// ---- FBs/Other Big Consumer/KNX/Linear/FB_OBC_Linear_KNX.TcPOU
FUNCTION_BLOCK FB_OBC_Linear_KNX
VAR_INPUT PERSISTENT
	bEnable									: BOOL;												//{#lynus.ag#()} //Enable the Fuctionblock and his logic
	bPowerDataInvers						: BOOL;												//With True its possible to invert all received power data from the electric meter
	bNoLinear								: BOOL;												//Output Power from the device is not linear. Use the Values from the Table Of Interpolation Points.
	diNrOfKNXMasterLine_IN					: DINT;												//Number of the KNX Master Function on what this function can receive or write data
	diNrOfEMS_IN							: DINT;												//Number of EMS what control this Device.
	diNrOfEM_IN_OBC							: DINT;												//Number of the electric meter for incoming power data. (Power Data for this Device)
	stSetupOBC								: ST_Setup_OBC;										//{#lynus.ag#()} //Setup other big consumer
	strGroupAddr							: EIB_GROUP_ADDR;									//KNX group address which should be controlled with this function
	arrTableOfInterpolationPoints			: ARRAY[1..10] OF REAL;								//Table Of Interpolation Points. Corresponds to the different power values in the non-linear curve of the device. The last value must correspond to the maximum power.
END_VAR
VAR_INPUT
END_VAR
VAR_OUTPUT
	stDataOBC								: ST_OBC_Output;									//{#lynus.ag#()} //Output Data other big consumer
	diNrOfOBC_OUT							: DINT;												//Active Number from the other big consumer for using on other functions
END_VAR
VAR
	{attribute 'hide'}
	fbOBC									: FB_BigConsumer;									//Function for other big consumer
	{attribute 'hide'}
	fbNumberDevice							: FB_NumberOfDevice;								//Function block to calcualte the number of the Device
	{attribute 'hide'}
	fbInterpolation							: FB_Lin_Interpolation;								//Function for interpolation
	fbDIExternalLock						: FB_XL1XXX_DI;										//Digital Input from external loock signal
	{attribute 'hide'}
	fbKNXSend								: EIB_2OCTET_FLOAT_SEND_EX;							//Function to send a Float value to the KNX Bus
	{attribute 'hide'}
	timDissableFunctions					: TON;												//Timer to dissable the Function after Lynus_Standards.Constants_General.tTimeDissableLynusFunctions Days without connection to the Lynus Cloud
	{attribute 'hide'}
	timResetConnectionOnGVL					: TON;												//Timer to try reset the connection Flag on the GVL. (When somebody delete the Connection Function and make only a onlinechange)
	{attribute 'hide'}
	arrPD									: ARRAY[1..27] OF FB_PersistentData_Number;			//Function to save persistent data 
	{attribute 'hide'}
	byWaitInStep							: BYTE;												//Wait in Step before start to clean data on PLC
	{attribute 'hide'}
	iStateGVLData							: INT;												//State machine to handle the data on the GVL
	{attribute 'hide'}
	diNumberOfActiveBatterys				: DINT;												//Number of active batterys
	{attribute 'hide'}
	diNumberOfBatteryInverterInEPO			: DINT;												//Number of battery inverters that work in Emergency Power operation 
	{attribute 'hide'}
	diCounterForGVL							: DINT;												//Counter to clean old data on GVL
	{attribute 'hide'}
	diLPForGVL								: DINT;												//Loop to clean old data on GVL
	{attribute 'hide'}
	dwSumSOC								: DWORD;											//Sum of the SOC from all batterys
	{attribute 'hide'}
	liLPBatteryData							: LINT;												//Loop to check some data from batterys
	{attribute 'hide'}
	liLPInEPO								: LINT;												//Loop to check if 1 or more battery inverters build a island grid	
END_VAR
VAR PERSISTENT
	{attribute 'conditionalshow'}
	diNrOfEMS_IN_CP							: DINT;												//Number of EMS what control this Device to compare with the original
END_VAR

//Creator : Kai Ebensperger
//Company : Lynus AG
//Date : 24.08.2021
//Version : 1.0.0.0

//With this function block its possible to control a other big consumer with the plc
//The output signal to control the big consumer is sending to the KNX Group Adress from the Inputs
//The value what is sending to the KNX Bus is between 0 and 100 to control the device.
//Also the Power Data can by displayed with this functionblock

//NOTE for diNr.....Designation => 
//_IN = Here Data come in from other Functions or go out to other functions about the GVL
//_OUT = Here Data go out to other functions about the GVL

(*------------------------------------------------------------Limits----------------------------------------------------------------------------------*)

diNrOfEMS_IN := LIMIT(0,diNrOfEMS_IN,Constants_Energy.diMaxNumberOfEMS);
	diNrOfEM_IN_OBC := LIMIT(0,diNrOfEM_IN_OBC,Constants_Energy.diMaxNumberOfElectricMeters);
		diNrOfKNXMasterLine_IN := LIMIT(0,diNrOfKNXMasterLine_IN,Constants_Bussystems.diMaxNumberOfKNXMasterKL6301);	

strGroupAddr.MAIN := LIMIT(0,strGroupAddr.MAIN,31);
	strGroupAddr.SUB_MAIN := LIMIT(0,strGroupAddr.SUB_MAIN,7);
			
(*------------------------------------------------------------------Power Data----------------------------------------------------------------------------*)

IF NOT bPowerDataInvers THEN
	fbOBC.lrCounterEnergyT1_Consumption := Lynus_Standards.GVL_Energy.stDataElectricMeters[diNrOfEM_IN_OBC].lrCounterEnergyT1_Production * 1000;
	fbOBC.lrCounterEnergyT2_Consumption := Lynus_Standards.GVL_Energy.stDataElectricMeters[diNrOfEM_IN_OBC].lrCounterEnergyT2_Production * 1000;
	fbOBC.lrCounterEnergyT1_Production := Lynus_Standards.GVL_Energy.stDataElectricMeters[diNrOfEM_IN_OBC].lrCounterEnergyT1_Consumption * 1000;
	fbOBC.lrCounterEnergyT2_Production := Lynus_Standards.GVL_Energy.stDataElectricMeters[diNrOfEM_IN_OBC].lrCounterEnergyT1_Consumption * 1000;
	fbOBC.lrTotalCounterEnergy_Consumption := Lynus_Standards.GVL_Energy.stDataElectricMeters[diNrOfEM_IN_OBC].lrTotalCounterEnergy_Production * 1000;
	fbOBC.lrTotalCounterEnergy_Production := Lynus_Standards.GVL_Energy.stDataElectricMeters[diNrOfEM_IN_OBC].lrTotalCounterEnergy_Consumption * 1000;
		fbOBC.lrPowerOBC := (Lynus_Standards.GVL_Energy.stDataElectricMeters[diNrOfEM_IN_OBC].lrPower * 1000) * - 1;
ELSE
	fbOBC.lrCounterEnergyT1_Consumption := Lynus_Standards.GVL_Energy.stDataElectricMeters[diNrOfEM_IN_OBC].lrCounterEnergyT1_Consumption * 1000;
	fbOBC.lrCounterEnergyT2_Consumption := Lynus_Standards.GVL_Energy.stDataElectricMeters[diNrOfEM_IN_OBC].lrCounterEnergyT2_Consumption * 1000;
	fbOBC.lrCounterEnergyT1_Production := Lynus_Standards.GVL_Energy.stDataElectricMeters[diNrOfEM_IN_OBC].lrCounterEnergyT1_Production * 1000;
	fbOBC.lrCounterEnergyT2_Production := Lynus_Standards.GVL_Energy.stDataElectricMeters[diNrOfEM_IN_OBC].lrCounterEnergyT2_Production * 1000;
	fbOBC.lrTotalCounterEnergy_Consumption := Lynus_Standards.GVL_Energy.stDataElectricMeters[diNrOfEM_IN_OBC].lrTotalCounterEnergy_Consumption * 1000;
	fbOBC.lrTotalCounterEnergy_Production := Lynus_Standards.GVL_Energy.stDataElectricMeters[diNrOfEM_IN_OBC].lrTotalCounterEnergy_Production * 1000;
		fbOBC.lrPowerOBC := Lynus_Standards.GVL_Energy.stDataElectricMeters[diNrOfEM_IN_OBC].lrPower * 1000;
END_IF

(*-------------------------------------------------------------Calcualte the number of OBC---------------------------------------------------------------*)

fbNumberDevice(
	diActualNumberOfDevices:= Lynus_Standards.GVL_Energy.stNumberOfDevices.diNumberOfOBC, 
	diMaxNumberOfDevices:= Constants_Energy.diMaxNumberOfOtherBigConsumers, 
	udiCounterOnlineChange:= TwinCAT_SystemInfoVarList._AppInfo.OnlineChangeCnt, 
	bNumberIsCalculatet=> , 
	bFPNumberIsCalculatet=> , 
	bOnlineChange=> , 
	diNumberForThisDevice=> diNrOfOBC_OUT, 
	diNumberOfTotalDevices=> );

//Write new Numer on GVL
IF fbNumberDevice.bFPNumberIsCalculatet THEN
	Lynus_Standards.GVL_Energy.stNumberOfDevices.diNumberOfOBC := fbNumberDevice.diNumberOfTotalDevices;	
END_IF 

//Delete old Number on GVL
IF fbNumberDevice.bOnlineChange THEN 
	Lynus_Standards.GVL_Energy.stNumberOfDevices.diNumberOfOBC := diNrOfOBC_OUT;	
		iStateGVLData := 1; 
END_IF

(*-------------------------------------------------------------Service from Backend is ready and check the connection to backen for dissabel/enable Function---------------------------------------------------------------*)

//Try to reset the variable for connection on the GVL. When all is normal then the Lynus Mqtt connection function set this variable to true in the next cycle
//When we have no connection to the backend then after Lynus_Standards.Constants_General.tTimeDissableLynusFunctions days the Function is dissabled with all of his functionalities
timResetConnectionOnGVL(IN:= NOT timResetConnectionOnGVL.Q, PT:= T#1H, Q=> , ET=> );
	IF timResetConnectionOnGVL.Q THEN Lynus_Standards.GVL_Communicator.bStateConnectionToEnableFunctions := FALSE; END_IF
		IF NOT Lynus_Standards.GVL_Communicator.bStateConnectionToEnableFunctions THEN timDissableFunctions.IN := TRUE; ELSE timDissableFunctions.IN := FALSE; END_IF  
			timDissableFunctions(IN:= , PT:= Lynus_Standards.Constants_General.tTimeDissableLynusFunctions, Q=> , ET=> );

(*------------------------------------------------------------------Error----------------------------------------------------------------------------*)

IF timDissableFunctions.Q THEN fbOBC.bWarning := TRUE; fbOBC.iWarningCode := 0; ELSE fbOBC.bWarning := FALSE; END_IF 
	IF Lynus_Standards.GVL_Energy.stNumberOfDevices.diNumberOfOBC > Constants_Energy.diMaxNumberOfOtherBigConsumers OR fbKNXSend.bError THEN 
		fbOBC.bError := TRUE;
	ELSE 
		fbOBC.bError := FALSE;
	END_IF 	
	
IF Lynus_Standards.GVL_Energy.stNumberOfDevices.diNumberOfOBC > Constants_Energy.diMaxNumberOfOtherBigConsumers THEN fbOBC.iErrorCode := 1;
ELSIF fbKNXSend.bError THEN fbOBC.iErrorCode := 0;
END_IF   	
	
(*------------------------------------------------------------------Logic----------------------------------------------------------------------------*)
	
//Calcualte the total SOC if we have more then 1 battery in our system
diNumberOfActiveBatterys := 0;
	dwSumSOC := 0;
		FOR liLPBatteryData := 1 TO Constants_Energy.diMaxNumberOfBatterys BY 1 DO
			IF Lynus_Standards.GVL_Energy.stDataOfBatterys[diNrOfEMS_IN,liLPBatteryData].bEnabled THEN diNumberOfActiveBatterys := diNumberOfActiveBatterys + 1; END_IF
				dwSumSOC := dwSumSOC + Lynus_Standards.GVL_Energy.stDataOfBatterys[diNrOfEMS_IN,liLPBatteryData].dwSOC;
		END_FOR
	
IF diNumberOfActiveBatterys > 0 THEN
	fbOBC.dwBatterySOC := DINT_TO_DWORD(DWORD_TO_DINT(dwSumSOC) / diNumberOfActiveBatterys);
ELSE
	fbOBC.dwBatterySOC := 100;	//When we have no battery in the ems system
END_IF

//Check if one or more Batterysystems or batteryinverter make island mode
diNumberOfBatteryInverterInEPO := 0;
	FOR liLPInEPO := 1 TO Constants_Energy.diMaxNumberOfBatteryInverters BY 1 DO
		IF Lynus_Standards.GVL_Energy.stDataOfBatteryInverters[diNrOfEMS_IN,liLPInEPO].bWorkOnIslandMode THEN fbOBC.bEPOIsActive := TRUE; diNumberOfBatteryInverterInEPO := diNumberOfBatteryInverterInEPO + 1; END_IF
	END_FOR 
		IF diNumberOfBatteryInverterInEPO <= 0 THEN fbOBC.bEPOIsActive := FALSE; END_IF

//Digital input for external lock signal
fbDIExternalLock(bInvers:= FALSE, bSignal=> );

fbOBC(
	bEnable:= bEnable AND NOT timDissableFunctions.Q,
	bError:= , 
	bEPOIsActive:= , 
	bExternalLock:= fbDIExternalLock.bSignal, 
	bWriteWithDelay:= TRUE, 
	iErrorCode:= , 
	iWarningCode:= , 
	dwBatterySOC:= , 
	lrTotalCounterEnergy_Consumption:= , 
	lrTotalCounterEnergy_Production:= , 
	lrCounterEnergyT1_Consumption:= , 
	lrCounterEnergyT2_Consumption:= , 
	lrCounterEnergyT1_Production:= , 
	lrCounterEnergyT2_Production:= , 
	lrPowerOBC:= , 
	rTargetPower:= Lynus_Standards.GVL_Energy.stDataOtherBigConsumers[diNrOfEMS_IN,diNrOfOBC_OUT].rTargetPowerEMS, 
	tTimDelayOutput:= T#5S, 
	stSetupOBC:= stSetupOBC, 
	stDataOBCOut=> , 
	stDataOBCOutDelay=> stDataOBC);											
	
(*-------------------------------------------------------------------------Output to KNX----------------------------------------------------------------------*)

IF bNoLinear THEN 
	fbInterpolation.rXInputValue := (stSetupOBC.rMaxPower * fbOBC.stDataOBCOut.rTargetPower) / 100; 
		fbInterpolation.arrYIntermediateValues[1] := 10;
			fbInterpolation.arrYIntermediateValues[2] := 20;
				fbInterpolation.arrYIntermediateValues[3] := 30;
					fbInterpolation.arrYIntermediateValues[4] := 40;
						fbInterpolation.arrYIntermediateValues[5] := 50;
	fbInterpolation.arrYIntermediateValues[6] := 60;
		fbInterpolation.arrYIntermediateValues[7] := 70;
			fbInterpolation.arrYIntermediateValues[8] := 80;
				fbInterpolation.arrYIntermediateValues[9] := 90;
					fbInterpolation.arrYIntermediateValues[10] := 100;
	fbInterpolation(rXInputValue:=, arrXIntermediateValues:= arrTableOfInterpolationPoints, arrYIntermediateValues:=, rYOutputValue=> );
END_IF

IF bNoLinear THEN 
	fbKNXSend.rData := fbInterpolation.rYOutputValue;
ELSE
	fbKNXSend.rData := fbOBC.stDataOBCOut.rTargetPower;
END_IF
	
fbKNXSend(
	bStart:= TRUE, 
	iMode:= 2, 
	CyclePolling:= T#200MS, 
	MinSendTime:= T#500MS, 
	Group_Address:= strGroupAddr, 
	rData:= , 
	str_Rec:= Lynus_Standards.GVL_Bussystems.stDataOfKNXMasterKL6301[diNrOfKNXMasterLine_IN], 
	bEnableReadReq:= FALSE, 
	bBusy=> , 
	bError=> , 
	iErrorID=> );

(*-----------------------------------------------------------Handle data to Global structure for the other big consumers-----------------------------------------------------------------*)

//Delte al old Data on GVL after a online change or change on the variable diNrOfEMS_IDOD
IF diNrOfEM_IN_OBC <> diNrOfEMS_IN_CP AND iStateGVLData = 0 THEN iStateGVLData := 10; END_IF 

CASE iStateGVLData OF
	
	0://Init Step
		byWaitInStep := 0;
			diCounterForGVL := 1;
	
	1://Wait for 4 Steps before clean al Data on GVL
		byWaitInStep := byWaitInStep + 1;
			IF byWaitInStep >= 4 AND fbNumberDevice.bNumberIsCalculatet THEN iStateGVLData := 2; END_IF
				//To much Devices, back to the Init step
				IF byWaitInStep >= 4 AND NOT fbNumberDevice.bNumberIsCalculatet THEN iStateGVLData := 0; END_IF	
			
	2://Clear all Data in GVL
		FOR diLPForGVL := 1 TO Constants_Energy.diMaxNumberOfEMS BY 1 DO 
			Lynus_Standards.GVL_Energy.stDataOtherBigConsumers[diLPForGVL,diCounterForGVL].bEnabled := FALSE;
				Lynus_Standards.GVL_Energy.stDataOtherBigConsumers[diLPForGVL,diCounterForGVL].bIsControllable := FALSE;
					Lynus_Standards.GVL_Energy.stDataOtherBigConsumers[diLPForGVL,diCounterForGVL].byPriority := 0;
						Lynus_Standards.GVL_Energy.stDataOtherBigConsumers[diLPForGVL,diCounterForGVL].byErrorWarning := 0;
							Lynus_Standards.GVL_Energy.stDataOtherBigConsumers[diLPForGVL,diCounterForGVL].lrPower := 0;
								Lynus_Standards.GVL_Energy.stDataOtherBigConsumers[diLPForGVL,diCounterForGVL].lrPowerConsumption := 0;
									Lynus_Standards.GVL_Energy.stDataOtherBigConsumers[diLPForGVL,diCounterForGVL].lrPowerProduction := 0;
										Lynus_Standards.GVL_Energy.stDataOtherBigConsumers[diLPForGVL,diCounterForGVL].rMaxPower := 0;
											//Set also the target value from ems back here to 0 and not in EMS function because EMS is in Standy when we have a online change (Problem when we delete a ems function and make a online change)
											Lynus_Standards.GVL_Energy.stDataOtherBigConsumers[diLPForGVL,diCounterForGVL].rTargetPowerEMS := 0;
		END_FOR
			diCounterForGVL := diCounterForGVL + 1;
				diCounterForGVL := LIMIT(0,diCounterForGVL,Constants_Energy.diMaxNumberOfOtherBigConsumers);
					//Back to the init step
					IF diCounterForGVL >= Constants_Energy.diMaxNumberOfOtherBigConsumers THEN iStateGVLData := 0; END_IF

	10://Clear old Data on GVL 	
		Lynus_Standards.GVL_Energy.stDataOtherBigConsumers[diNrOfEMS_IN_CP,diNrOfOBC_OUT].bEnabled := FALSE;
			Lynus_Standards.GVL_Energy.stDataOtherBigConsumers[diNrOfEMS_IN_CP,diNrOfOBC_OUT].bIsControllable := FALSE;
				Lynus_Standards.GVL_Energy.stDataOtherBigConsumers[diNrOfEMS_IN_CP,diNrOfOBC_OUT].byPriority := 0;
					Lynus_Standards.GVL_Energy.stDataOtherBigConsumers[diNrOfEMS_IN_CP,diNrOfOBC_OUT].byErrorWarning := 0;
						Lynus_Standards.GVL_Energy.stDataOtherBigConsumers[diNrOfEMS_IN_CP,diNrOfOBC_OUT].lrPower := 0;
							Lynus_Standards.GVL_Energy.stDataOtherBigConsumers[diNrOfEMS_IN_CP,diNrOfOBC_OUT].lrPowerConsumption := 0;
								Lynus_Standards.GVL_Energy.stDataOtherBigConsumers[diNrOfEMS_IN_CP,diNrOfOBC_OUT].lrPowerProduction := 0;
									Lynus_Standards.GVL_Energy.stDataOtherBigConsumers[diNrOfEMS_IN_CP,diNrOfOBC_OUT].rMaxPower := 0;
	
		diNrOfEMS_IN_CP := diNrOfEMS_IN;
			//Back to the init step
			iStateGVLData := 0;

END_CASE 	 

IF diNrOfOBC_OUT > 0 AND fbNumberDevice.bNumberIsCalculatet AND diNrOfEMS_IN > 0 THEN
	Lynus_Standards.GVL_Energy.stDataOtherBigConsumers[diNrOfEMS_IN,diNrOfOBC_OUT].bEnabled := fbOBC.stDataOBCOut.bEnabled;
		Lynus_Standards.GVL_Energy.stDataOtherBigConsumers[diNrOfEMS_IN,diNrOfOBC_OUT].bIsControllable := TRUE;
			Lynus_Standards.GVL_Energy.stDataOtherBigConsumers[diNrOfEMS_IN,diNrOfOBC_OUT].byPriority := fbOBC.stDataOBCOut.byPriority;
				Lynus_Standards.GVL_Energy.stDataOtherBigConsumers[diNrOfEMS_IN,diNrOfOBC_OUT].byErrorWarning := fbOBC.stDataOBCOut.byErrorWarning;
					Lynus_Standards.GVL_Energy.stDataOtherBigConsumers[diNrOfEMS_IN,diNrOfOBC_OUT].lrPower := fbOBC.stDataOBCOut.lrPower;
						Lynus_Standards.GVL_Energy.stDataOtherBigConsumers[diNrOfEMS_IN,diNrOfOBC_OUT].lrPowerConsumption := fbOBC.stDataOBCOut.lrPowerConsumption;
							Lynus_Standards.GVL_Energy.stDataOtherBigConsumers[diNrOfEMS_IN,diNrOfOBC_OUT].lrPowerProduction := fbOBC.stDataOBCOut.lrPowerProduction;
								Lynus_Standards.GVL_Energy.stDataOtherBigConsumers[diNrOfEMS_IN,diNrOfOBC_OUT].rMaxPower := fbOBC.stDataOBCOut.rMaxPower;
END_IF

(*----------------------------------------------------------Save persistent data----------------------------------------------------------------*)

arrPD[1](lrValue:= BOOL_TO_LREAL(bEnable), bEventBasedActive=> );
arrPD[2](lrValue:= BOOL_TO_LREAL(bPowerDataInvers), bEventBasedActive=> );
arrPD[3](lrValue:= DINT_TO_LREAL(diNrOfEMS_IN), bEventBasedActive=> );
arrPD[4](lrValue:= DINT_TO_LREAL(diNrOfEM_IN_OBC), bEventBasedActive=> );
arrPD[5](lrValue:= DINT_TO_LREAL(diNrOfEMS_IN_CP), bEventBasedActive=> );
arrPD[6](lrValue:= BOOL_TO_LREAL(stSetupOBC.bManualyOn), bEventBasedActive=> );
arrPD[7](lrValue:= BOOL_TO_LREAL(stSetupOBC.bOnEmergPowerOff), bEventBasedActive=> );
arrPD[8](lrValue:= BYTE_TO_LREAL(stSetupOBC.byDisableSOC), bEventBasedActive=> );
arrPD[9](lrValue:= BYTE_TO_LREAL(stSetupOBC.byEnableSOC), bEventBasedActive=> );
arrPD[10](lrValue:= BYTE_TO_LREAL(stSetupOBC.byManualyTargetPower), bEventBasedActive=> );
arrPD[11](lrValue:= BYTE_TO_LREAL(stSetupOBC.byPriority), bEventBasedActive=> );
arrPD[12](lrValue:= REAL_TO_LREAL(stSetupOBC.rMaxPower), bEventBasedActive=> );
arrPD[13](lrValue:= DINT_TO_LREAL(diNrOfKNXMasterLine_IN), bEventBasedActive=> );
arrPD[14](lrValue:= BYTE_TO_LREAL(strGroupAddr.MAIN), bEventBasedActive=> );
arrPD[15](lrValue:= BYTE_TO_LREAL(strGroupAddr.NUMBER), bEventBasedActive=> );
arrPD[16](lrValue:= BYTE_TO_LREAL(strGroupAddr.SUB_MAIN), bEventBasedActive=> );
arrPD[17](lrValue:= BOOL_TO_LREAL(bNoLinear), bEventBasedActive=> );
arrPD[18](lrValue:= REAL_TO_LREAL(arrTableOfInterpolationPoints[1]), bEventBasedActive=> );
arrPD[19](lrValue:= REAL_TO_LREAL(arrTableOfInterpolationPoints[2]), bEventBasedActive=> );
arrPD[20](lrValue:= REAL_TO_LREAL(arrTableOfInterpolationPoints[3]), bEventBasedActive=> );
arrPD[21](lrValue:= REAL_TO_LREAL(arrTableOfInterpolationPoints[4]), bEventBasedActive=> );
arrPD[22](lrValue:= REAL_TO_LREAL(arrTableOfInterpolationPoints[5]), bEventBasedActive=> );
arrPD[23](lrValue:= REAL_TO_LREAL(arrTableOfInterpolationPoints[6]), bEventBasedActive=> );
arrPD[24](lrValue:= REAL_TO_LREAL(arrTableOfInterpolationPoints[7]), bEventBasedActive=> );
arrPD[25](lrValue:= REAL_TO_LREAL(arrTableOfInterpolationPoints[8]), bEventBasedActive=> );
arrPD[26](lrValue:= REAL_TO_LREAL(arrTableOfInterpolationPoints[9]), bEventBasedActive=> );
arrPD[27](lrValue:= REAL_TO_LREAL(arrTableOfInterpolationPoints[10]), bEventBasedActive=> );

END_FUNCTION_BLOCK

// ---- FBs/Other Big Consumer/KNX/OnOff/FB_OBC_OnOff_KNX.TcPOU
FUNCTION_BLOCK FB_OBC_OnOff_KNX
VAR_INPUT PERSISTENT
	bEnable									: BOOL;												//{#lynus.ag#()} //Enable the Fuctionblock and his logic
	bPowerDataInvers						: BOOL;												//With True its possible to invert all received power data from the electric meter
	diNrOfKNXMasterLine_IN					: DINT;												//Number of the KNX Master Function on what this function can receive or write data
	diNrOfEMS_IN							: DINT;												//Number of EMS what control this Device.
	diNrOfEM_IN_OBC							: DINT;												//Number of the electric meter for incoming power data. (Power Data for this Device)
	stSetupOBC								: ST_Setup_OBC;										//{#lynus.ag#()} //Setup other big consumer
	strGroupAddr							: EIB_GROUP_ADDR;									//KNX group address which should be controlled with this function
END_VAR
VAR_INPUT
END_VAR
VAR_OUTPUT
	stDataOBC								: ST_OBC_Output;									//{#lynus.ag#()} //Output Data other big consumer
	diNrOfOBC_OUT							: DINT;												//Active Number from the other big consumer for using on other functions
END_VAR
VAR
	{attribute 'hide'}
	fbOBC									: FB_BigConsumer;									//Function for other big consumer
	{attribute 'hide'}
	fbNumberDevice							: FB_NumberOfDevice;								//Function block to calcualte the number of the Device
	fbDIExternalLock						: FB_XL1XXX_DI;										//Digital Input from external loock signal
	{attribute 'hide'}
	fbKNXSend								: EIB_BIT_SEND_EX;									//Function to send a Float value to the KNX Bus
	{attribute 'hide'}
	timDissableFunctions					: TON;												//Timer to dissable the Function after Lynus_Standards.Constants_General.tTimeDissableLynusFunctions Days without connection to the Lynus Cloud
	{attribute 'hide'}
	timResetConnectionOnGVL					: TON;												//Timer to try reset the connection Flag on the GVL. (When somebody delete the Connection Function and make only a onlinechange)
	{attribute 'hide'}
	arrPD									: ARRAY[1..16] OF FB_PersistentData_Number;			//Function to save persistent data 
	{attribute 'hide'}
	byWaitInStep							: BYTE;												//Wait in Step before start to clean data on PLC
	{attribute 'hide'}
	iStateGVLData							: INT;												//State machine to handle the data on the GVL
	{attribute 'hide'}
	diNumberOfActiveBatterys				: DINT;												//Number of active batterys
	{attribute 'hide'}
	diNumberOfBatteryInverterInEPO			: DINT;												//Number of battery inverters that work in Emergency Power operation 
	{attribute 'hide'}
	diCounterForGVL							: DINT;												//Counter to clean old data on GVL
	{attribute 'hide'}
	diLPForGVL								: DINT;												//Loop to clean old data on GVL
	{attribute 'hide'}
	dwSumSOC								: DWORD;											//Sum of the SOC from all batterys
	{attribute 'hide'}
	liLPBatteryData							: LINT;												//Loop to check some data from batterys
	{attribute 'hide'}
	liLPInEPO								: LINT;												//Loop to check if 1 or more battery inverters build a island grid	
END_VAR
VAR PERSISTENT
	{attribute 'conditionalshow'}
	diNrOfEMS_IN_CP							: DINT;												//Number of EMS what control this Device to compare with the original
END_VAR

//Creator : Kai Ebensperger
//Company : Lynus AG
//Date : 24.08.2021
//Version : 1.0.0.0

//With this function block its possible to control a other big consumer with the plc
//The output signal to control the big consumer is sending to the KNX Group Adress from the Inputs
//The value what is sending to the KNX Bus is 0 to switch off or 1 to switch on.
//Also the Power Data can by displayed with this functionblock

//NOTE for diNr.....Designation => 
//_IN = Here Data come in from other Functions or go out to other functions about the GVL
//_OUT = Here Data go out to other functions about the GVL

(*------------------------------------------------------------Limits----------------------------------------------------------------------------------*)

diNrOfEMS_IN := LIMIT(0,diNrOfEMS_IN,Constants_Energy.diMaxNumberOfEMS);
	diNrOfEM_IN_OBC := LIMIT(0,diNrOfEM_IN_OBC,Constants_Energy.diMaxNumberOfElectricMeters);
		diNrOfKNXMasterLine_IN := LIMIT(0,diNrOfKNXMasterLine_IN,Constants_Bussystems.diMaxNumberOfKNXMasterKL6301);	

strGroupAddr.MAIN := LIMIT(0,strGroupAddr.MAIN,31);
	strGroupAddr.SUB_MAIN := LIMIT(0,strGroupAddr.SUB_MAIN,7);
			
(*------------------------------------------------------------------Power Data----------------------------------------------------------------------------*)

IF NOT bPowerDataInvers THEN
	fbOBC.lrCounterEnergyT1_Consumption := Lynus_Standards.GVL_Energy.stDataElectricMeters[diNrOfEM_IN_OBC].lrCounterEnergyT1_Production * 1000;
	fbOBC.lrCounterEnergyT2_Consumption := Lynus_Standards.GVL_Energy.stDataElectricMeters[diNrOfEM_IN_OBC].lrCounterEnergyT2_Production * 1000;
	fbOBC.lrCounterEnergyT1_Production := Lynus_Standards.GVL_Energy.stDataElectricMeters[diNrOfEM_IN_OBC].lrCounterEnergyT1_Consumption * 1000;
	fbOBC.lrCounterEnergyT2_Production := Lynus_Standards.GVL_Energy.stDataElectricMeters[diNrOfEM_IN_OBC].lrCounterEnergyT1_Consumption * 1000;
	fbOBC.lrTotalCounterEnergy_Consumption := Lynus_Standards.GVL_Energy.stDataElectricMeters[diNrOfEM_IN_OBC].lrTotalCounterEnergy_Production * 1000;
	fbOBC.lrTotalCounterEnergy_Production := Lynus_Standards.GVL_Energy.stDataElectricMeters[diNrOfEM_IN_OBC].lrTotalCounterEnergy_Consumption * 1000;
		fbOBC.lrPowerOBC := (Lynus_Standards.GVL_Energy.stDataElectricMeters[diNrOfEM_IN_OBC].lrPower * 1000) * - 1;
ELSE
	fbOBC.lrCounterEnergyT1_Consumption := Lynus_Standards.GVL_Energy.stDataElectricMeters[diNrOfEM_IN_OBC].lrCounterEnergyT1_Consumption * 1000;
	fbOBC.lrCounterEnergyT2_Consumption := Lynus_Standards.GVL_Energy.stDataElectricMeters[diNrOfEM_IN_OBC].lrCounterEnergyT2_Consumption * 1000;
	fbOBC.lrCounterEnergyT1_Production := Lynus_Standards.GVL_Energy.stDataElectricMeters[diNrOfEM_IN_OBC].lrCounterEnergyT1_Production * 1000;
	fbOBC.lrCounterEnergyT2_Production := Lynus_Standards.GVL_Energy.stDataElectricMeters[diNrOfEM_IN_OBC].lrCounterEnergyT2_Production * 1000;
	fbOBC.lrTotalCounterEnergy_Consumption := Lynus_Standards.GVL_Energy.stDataElectricMeters[diNrOfEM_IN_OBC].lrTotalCounterEnergy_Consumption * 1000;
	fbOBC.lrTotalCounterEnergy_Production := Lynus_Standards.GVL_Energy.stDataElectricMeters[diNrOfEM_IN_OBC].lrTotalCounterEnergy_Production * 1000;
		fbOBC.lrPowerOBC := Lynus_Standards.GVL_Energy.stDataElectricMeters[diNrOfEM_IN_OBC].lrPower * 1000;
END_IF

(*-------------------------------------------------------------Calcualte the number of OBC---------------------------------------------------------------*)

fbNumberDevice(
	diActualNumberOfDevices:= Lynus_Standards.GVL_Energy.stNumberOfDevices.diNumberOfOBC, 
	diMaxNumberOfDevices:= Constants_Energy.diMaxNumberOfOtherBigConsumers, 
	udiCounterOnlineChange:= TwinCAT_SystemInfoVarList._AppInfo.OnlineChangeCnt, 
	bNumberIsCalculatet=> , 
	bFPNumberIsCalculatet=> , 
	bOnlineChange=> , 
	diNumberForThisDevice=> diNrOfOBC_OUT, 
	diNumberOfTotalDevices=> );

//Write new Numer on GVL
IF fbNumberDevice.bFPNumberIsCalculatet THEN
	Lynus_Standards.GVL_Energy.stNumberOfDevices.diNumberOfOBC := fbNumberDevice.diNumberOfTotalDevices;	
END_IF 

//Delete old Number on GVL
IF fbNumberDevice.bOnlineChange THEN 
	Lynus_Standards.GVL_Energy.stNumberOfDevices.diNumberOfOBC := diNrOfOBC_OUT;	
		iStateGVLData := 1; 
END_IF

(*-------------------------------------------------------------Service from Backend is ready and check the connection to backen for dissabel/enable Function---------------------------------------------------------------*)

//Try to reset the variable for connection on the GVL. When all is normal then the Lynus Mqtt connection function set this variable to true in the next cycle
//When we have no connection to the backend then after Lynus_Standards.Constants_General.tTimeDissableLynusFunctions days the Function is dissabled with all of his functionalities
timResetConnectionOnGVL(IN:= NOT timResetConnectionOnGVL.Q, PT:= T#1H, Q=> , ET=> );
	IF timResetConnectionOnGVL.Q THEN Lynus_Standards.GVL_Communicator.bStateConnectionToEnableFunctions := FALSE; END_IF
		IF NOT Lynus_Standards.GVL_Communicator.bStateConnectionToEnableFunctions THEN timDissableFunctions.IN := TRUE; ELSE timDissableFunctions.IN := FALSE; END_IF  
			timDissableFunctions(IN:= , PT:= Lynus_Standards.Constants_General.tTimeDissableLynusFunctions, Q=> , ET=> );

(*------------------------------------------------------------------Error----------------------------------------------------------------------------*)

IF timDissableFunctions.Q THEN fbOBC.bWarning := TRUE; fbOBC.iWarningCode := 0; ELSE fbOBC.bWarning := FALSE; END_IF 
	IF Lynus_Standards.GVL_Energy.stNumberOfDevices.diNumberOfOBC > Constants_Energy.diMaxNumberOfOtherBigConsumers OR fbKNXSend.bError THEN 
		fbOBC.bError := TRUE;
	ELSE 
		fbOBC.bError := FALSE;
	END_IF 	
	
IF Lynus_Standards.GVL_Energy.stNumberOfDevices.diNumberOfOBC > Constants_Energy.diMaxNumberOfOtherBigConsumers THEN fbOBC.iErrorCode := 1;
ELSIF fbKNXSend.bError THEN fbOBC.iErrorCode := 0;
END_IF   	
	
(*------------------------------------------------------------------Logic----------------------------------------------------------------------------*)
	
//Calcualte the total SOC if we have more then 1 battery in our system
diNumberOfActiveBatterys := 0;
	dwSumSOC := 0;
		FOR liLPBatteryData := 1 TO Constants_Energy.diMaxNumberOfBatterys BY 1 DO
			IF Lynus_Standards.GVL_Energy.stDataOfBatterys[diNrOfEMS_IN,liLPBatteryData].bEnabled THEN diNumberOfActiveBatterys := diNumberOfActiveBatterys + 1; END_IF
				dwSumSOC := dwSumSOC + Lynus_Standards.GVL_Energy.stDataOfBatterys[diNrOfEMS_IN,liLPBatteryData].dwSOC;
		END_FOR
	
IF diNumberOfActiveBatterys > 0 THEN
	fbOBC.dwBatterySOC := DINT_TO_DWORD(DWORD_TO_DINT(dwSumSOC) / diNumberOfActiveBatterys);
ELSE
	fbOBC.dwBatterySOC := 100;	//When we have no battery in the ems system
END_IF

//Check if one or more Batterysystems or batteryinverter make island mode
diNumberOfBatteryInverterInEPO := 0;
	FOR liLPInEPO := 1 TO Constants_Energy.diMaxNumberOfBatteryInverters BY 1 DO
		IF Lynus_Standards.GVL_Energy.stDataOfBatteryInverters[diNrOfEMS_IN,liLPInEPO].bWorkOnIslandMode THEN fbOBC.bEPOIsActive := TRUE; diNumberOfBatteryInverterInEPO := diNumberOfBatteryInverterInEPO + 1; END_IF
	END_FOR 
		IF diNumberOfBatteryInverterInEPO <= 0 THEN fbOBC.bEPOIsActive := FALSE; END_IF

//Digital input for external lock signal
fbDIExternalLock(bInvers:= FALSE, bSignal=> );

//Functionblock OBC
fbOBC.stSetupOBC.bManualyOn := stSetupOBC.bManualyOn;
	IF fbOBC.stSetupOBC.bManualyOn THEN fbOBC.stSetupOBC.byManualyTargetPower := 100; ELSE fbOBC.stSetupOBC.byManualyTargetPower := 0; END_IF
		fbOBC.stSetupOBC.bOnEmergPowerOff := stSetupOBC.bOnEmergPowerOff;
			fbOBC.stSetupOBC.byDisableSOC := stSetupOBC.byDisableSOC;
				fbOBC.stSetupOBC.byEnableSOC := stSetupOBC.byEnableSOC;
					fbOBC.stSetupOBC.byPriority := stSetupOBC.byPriority;
						fbOBC.stSetupOBC.rMaxPower := stSetupOBC.rMaxPower;	

fbOBC(
	bEnable:= bEnable AND NOT timDissableFunctions.Q,
	bError:= , 
	bEPOIsActive:= , 
	bExternalLock:= fbDIExternalLock.bSignal, 
	bWriteWithDelay:= TRUE, 
	iErrorCode:= , 
	iWarningCode:= , 
	dwBatterySOC:= , 
	lrTotalCounterEnergy_Consumption:= , 
	lrTotalCounterEnergy_Production:= , 
	lrCounterEnergyT1_Consumption:= , 
	lrCounterEnergyT2_Consumption:= , 
	lrCounterEnergyT1_Production:= , 
	lrCounterEnergyT2_Production:= , 
	lrPowerOBC:= , 
	rTargetPower:= Lynus_Standards.GVL_Energy.stDataOtherBigConsumers[diNrOfEMS_IN,diNrOfOBC_OUT].rTargetPowerEMS, 
	tTimDelayOutput:= T#5S, 
	stSetupOBC:= , 
	stDataOBCOut=> , 
	stDataOBCOutDelay=> stDataOBC);											
	
(*-------------------------------------------------------------------------Output to KNX----------------------------------------------------------------------*)

IF fbOBC.stDataOBCOut.rTargetPower >= 100 THEN fbKNXSend.bData := TRUE; ELSE fbKNXSend.bData := FALSE; END_IF  
	
fbKNXSend(
	bStart:= TRUE, 
	iMode:= 2, 
	CyclePolling:= T#200MS, 
	MinSendTime:= T#500MS, 
	Group_Address:= strGroupAddr, 
	bData:= , 
	str_Rec:= Lynus_Standards.GVL_Bussystems.stDataOfKNXMasterKL6301[diNrOfKNXMasterLine_IN], 
	bEnableReadReq:= FALSE, 
	bBusy=> , 
	bError=> , 
	iErrorID=> );

(*-----------------------------------------------------------Handle data to Global structure for the other big consumers-----------------------------------------------------------------*)

//Delte al old Data on GVL after a online change or change on the variable diNrOfEMS_IDOD
IF diNrOfEM_IN_OBC <> diNrOfEMS_IN_CP AND iStateGVLData = 0 THEN iStateGVLData := 10; END_IF 

CASE iStateGVLData OF
	
	0://Init Step
		byWaitInStep := 0;
			diCounterForGVL := 1;
	
	1://Wait for 4 Steps before clean al Data on GVL
		byWaitInStep := byWaitInStep + 1;
			IF byWaitInStep >= 4 AND fbNumberDevice.bNumberIsCalculatet THEN iStateGVLData := 2; END_IF
				//To much Devices, back to the Init step
				IF byWaitInStep >= 4 AND NOT fbNumberDevice.bNumberIsCalculatet THEN iStateGVLData := 0; END_IF	
			
	2://Clear all Data in GVL
		FOR diLPForGVL := 1 TO Constants_Energy.diMaxNumberOfEMS BY 1 DO 
			Lynus_Standards.GVL_Energy.stDataOtherBigConsumers[diLPForGVL,diCounterForGVL].bEnabled := FALSE;
				Lynus_Standards.GVL_Energy.stDataOtherBigConsumers[diLPForGVL,diCounterForGVL].bIsControllable := FALSE;
					Lynus_Standards.GVL_Energy.stDataOtherBigConsumers[diLPForGVL,diCounterForGVL].byPriority := 0;
						Lynus_Standards.GVL_Energy.stDataOtherBigConsumers[diLPForGVL,diCounterForGVL].byErrorWarning := 0;
							Lynus_Standards.GVL_Energy.stDataOtherBigConsumers[diLPForGVL,diCounterForGVL].lrPower := 0;
								Lynus_Standards.GVL_Energy.stDataOtherBigConsumers[diLPForGVL,diCounterForGVL].lrPowerConsumption := 0;
									Lynus_Standards.GVL_Energy.stDataOtherBigConsumers[diLPForGVL,diCounterForGVL].lrPowerProduction := 0;
										Lynus_Standards.GVL_Energy.stDataOtherBigConsumers[diLPForGVL,diCounterForGVL].rMaxPower := 0;
											//Set also the target value from ems back here to 0 and not in EMS function because EMS is in Standy when we have a online change (Problem when we delete a ems function and make a online change)
											Lynus_Standards.GVL_Energy.stDataOtherBigConsumers[diLPForGVL,diCounterForGVL].rTargetPowerEMS := 0;
		END_FOR
			diCounterForGVL := diCounterForGVL + 1;
				diCounterForGVL := LIMIT(0,diCounterForGVL,Constants_Energy.diMaxNumberOfOtherBigConsumers);
					//Back to the init step
					IF diCounterForGVL >= Constants_Energy.diMaxNumberOfOtherBigConsumers THEN iStateGVLData := 0; END_IF

	10://Clear old Data on GVL 	
		Lynus_Standards.GVL_Energy.stDataOtherBigConsumers[diNrOfEMS_IN_CP,diNrOfOBC_OUT].bEnabled := FALSE;
			Lynus_Standards.GVL_Energy.stDataOtherBigConsumers[diNrOfEMS_IN_CP,diNrOfOBC_OUT].bIsControllable := FALSE;
				Lynus_Standards.GVL_Energy.stDataOtherBigConsumers[diNrOfEMS_IN_CP,diNrOfOBC_OUT].byPriority := 0;
					Lynus_Standards.GVL_Energy.stDataOtherBigConsumers[diNrOfEMS_IN_CP,diNrOfOBC_OUT].byErrorWarning := 0;
						Lynus_Standards.GVL_Energy.stDataOtherBigConsumers[diNrOfEMS_IN_CP,diNrOfOBC_OUT].lrPower := 0;
							Lynus_Standards.GVL_Energy.stDataOtherBigConsumers[diNrOfEMS_IN_CP,diNrOfOBC_OUT].lrPowerConsumption := 0;
								Lynus_Standards.GVL_Energy.stDataOtherBigConsumers[diNrOfEMS_IN_CP,diNrOfOBC_OUT].lrPowerProduction := 0;
									Lynus_Standards.GVL_Energy.stDataOtherBigConsumers[diNrOfEMS_IN_CP,diNrOfOBC_OUT].rMaxPower := 0;
	
		diNrOfEMS_IN_CP := diNrOfEMS_IN;
			//Back to the init step
			iStateGVLData := 0;

END_CASE 	 

IF diNrOfOBC_OUT > 0 AND fbNumberDevice.bNumberIsCalculatet AND diNrOfEMS_IN > 0 THEN
	Lynus_Standards.GVL_Energy.stDataOtherBigConsumers[diNrOfEMS_IN,diNrOfOBC_OUT].bEnabled := fbOBC.stDataOBCOut.bEnabled;
		Lynus_Standards.GVL_Energy.stDataOtherBigConsumers[diNrOfEMS_IN,diNrOfOBC_OUT].bIsControllable := FALSE;
			Lynus_Standards.GVL_Energy.stDataOtherBigConsumers[diNrOfEMS_IN,diNrOfOBC_OUT].byPriority := fbOBC.stDataOBCOut.byPriority;
				Lynus_Standards.GVL_Energy.stDataOtherBigConsumers[diNrOfEMS_IN,diNrOfOBC_OUT].byErrorWarning := fbOBC.stDataOBCOut.byErrorWarning;
					Lynus_Standards.GVL_Energy.stDataOtherBigConsumers[diNrOfEMS_IN,diNrOfOBC_OUT].lrPower := fbOBC.stDataOBCOut.lrPower;
						Lynus_Standards.GVL_Energy.stDataOtherBigConsumers[diNrOfEMS_IN,diNrOfOBC_OUT].lrPowerConsumption := fbOBC.stDataOBCOut.lrPowerConsumption;
							Lynus_Standards.GVL_Energy.stDataOtherBigConsumers[diNrOfEMS_IN,diNrOfOBC_OUT].lrPowerProduction := fbOBC.stDataOBCOut.lrPowerProduction;
								Lynus_Standards.GVL_Energy.stDataOtherBigConsumers[diNrOfEMS_IN,diNrOfOBC_OUT].rMaxPower := fbOBC.stDataOBCOut.rMaxPower;
END_IF

(*----------------------------------------------------------Save persistent data----------------------------------------------------------------*)

arrPD[1](lrValue:= BOOL_TO_LREAL(bEnable), bEventBasedActive=> );
arrPD[2](lrValue:= BOOL_TO_LREAL(bPowerDataInvers), bEventBasedActive=> );
arrPD[3](lrValue:= DINT_TO_LREAL(diNrOfEMS_IN), bEventBasedActive=> );
arrPD[4](lrValue:= DINT_TO_LREAL(diNrOfEM_IN_OBC), bEventBasedActive=> );
arrPD[5](lrValue:= DINT_TO_LREAL(diNrOfEMS_IN_CP), bEventBasedActive=> );
arrPD[6](lrValue:= BOOL_TO_LREAL(stSetupOBC.bManualyOn), bEventBasedActive=> );
arrPD[7](lrValue:= BOOL_TO_LREAL(stSetupOBC.bOnEmergPowerOff), bEventBasedActive=> );
arrPD[8](lrValue:= BYTE_TO_LREAL(stSetupOBC.byDisableSOC), bEventBasedActive=> );
arrPD[9](lrValue:= BYTE_TO_LREAL(stSetupOBC.byEnableSOC), bEventBasedActive=> );
arrPD[10](lrValue:= BYTE_TO_LREAL(stSetupOBC.byManualyTargetPower), bEventBasedActive=> );
arrPD[11](lrValue:= BYTE_TO_LREAL(stSetupOBC.byPriority), bEventBasedActive=> );
arrPD[12](lrValue:= REAL_TO_LREAL(stSetupOBC.rMaxPower), bEventBasedActive=> );
arrPD[13](lrValue:= DINT_TO_LREAL(diNrOfKNXMasterLine_IN), bEventBasedActive=> );
arrPD[14](lrValue:= BYTE_TO_LREAL(strGroupAddr.MAIN), bEventBasedActive=> );
arrPD[15](lrValue:= BYTE_TO_LREAL(strGroupAddr.NUMBER), bEventBasedActive=> );
arrPD[16](lrValue:= BYTE_TO_LREAL(strGroupAddr.SUB_MAIN), bEventBasedActive=> );

END_FUNCTION_BLOCK

// ---- FBs/Other Big Consumer/Linear AO/FB_OBC_Linear_AO.TcPOU
FUNCTION_BLOCK FB_OBC_Linear_AO
VAR_INPUT PERSISTENT
	bEnable									: BOOL;												//{#lynus.ag#()} //Enable the Fuctionblock and his logic
	bPowerDataInvers						: BOOL;												//With True its possible to invert all received power data from the electric meter
	bNoLinear								: BOOL;												//Output Power from the device is not linear. Use the Values from the Table Of Interpolation Points.
	diNrOfEMS_IN							: DINT;												//Number of EMS what control this Device.
	diNrOfEM_IN_OBC							: DINT;												//Number of the electric meter for incoming power data. (Power Data for this Device)
	stSetupOBC								: ST_Setup_OBC;										//{#lynus.ag#()} //Setup other big consumer
	arrTableOfInterpolationPoints			: ARRAY[1..10] OF REAL;								//Table Of Interpolation Points. Corresponds to the different power values in the non-linear curve of the device. The last value must correspond to the maximum power.
END_VAR
VAR_INPUT
END_VAR
VAR_OUTPUT
	stDataOBC								: ST_OBC_Output;									//{#lynus.ag#()} //Output Data other big consumer
	diNrOfOBC_OUT							: DINT;												//Active Number from the other big consumer for using on other functions
	rTargetPowerForExtFunc					: REAL;												//Target Power from 0% to +100% to use on a external Function
END_VAR
VAR
	{attribute 'hide'}
	fbOBC									: FB_BigConsumer;									//Function for other big consumer
	{attribute 'hide'}
	fbNumberDevice							: FB_NumberOfDevice;								//Function block to calcualte the number of the Device
	{attribute 'hide'}
	fbInterpolation							: FB_Lin_Interpolation;								//Function for interpolation
	fbDIExternalLock						: FB_XL1XXX_DI;										//Digital Input from external loock signal
	fbAOOBC									: FB_XL4XXX_AO;										//Analog Output to swtich on and off and controll the OBC
	{attribute 'hide'}
	timDissableFunctions					: TON;												//Timer to dissable the Function after Lynus_Standards.Constants_General.tTimeDissableLynusFunctions Days without connection to the Lynus Cloud
	{attribute 'hide'}
	timResetConnectionOnGVL					: TON;												//Timer to try reset the connection Flag on the GVL. (When somebody delete the Connection Function and make only a onlinechange)
	{attribute 'hide'}
	arrPD									: ARRAY[1..23] OF FB_PersistentData_Number;			//Function to save persistent data 
	{attribute 'hide'}
	byWaitInStep							: BYTE;												//Wait in Step before start to clean data on PLC
	{attribute 'hide'}
	iStateGVLData							: INT;												//State machine to handle the data on the GVL
	{attribute 'hide'}
	diNumberOfActiveBatterys				: DINT;												//Number of active batterys
	{attribute 'hide'}
	diNumberOfBatteryInverterInEPO			: DINT;												//Number of battery inverters that work in Emergency Power operation 
	{attribute 'hide'}
	diCounterForGVL							: DINT;												//Counter to clean old data on GVL
	{attribute 'hide'}
	diLPForGVL								: DINT;												//Loop to clean old data on GVL
	{attribute 'hide'}
	dwSumSOC								: DWORD;											//Sum of the SOC from all batterys
	{attribute 'hide'}
	liLPBatteryData							: LINT;												//Loop to check some data from batterys
	{attribute 'hide'}
	liLPInEPO								: LINT;												//Loop to check if 1 or more battery inverters build a island grid	
END_VAR
VAR PERSISTENT
	{attribute 'conditionalshow'}
	diNrOfEMS_IN_CP							: DINT;												//Number of EMS what control this Device to compare with the original
END_VAR

//Creator : Kai Ebensperger
//Company : Lynus AG
//Date : 19.05.2021
//Version : 1.0.0.0

//With this function block its possible to control a other big consumer with the plc
//The output signal to control the big consumer is a analog output signal (0-10V or 4-20mA)
//With this function block its possible to control the OBC with a target power value over the analog signal. The output signal is linear
//Also the Power Data can by displayed with this functionblock

//NOTE for diNr.....Designation => 
//_IN = Here Data come in from other Functions or go out to other functions about the GVL
//_OUT = Here Data go out to other functions about the GVL

(*------------------------------------------------------------Limits----------------------------------------------------------------------------------*)

diNrOfEMS_IN := LIMIT(0,diNrOfEMS_IN,Constants_Energy.diMaxNumberOfEMS);
	diNrOfEM_IN_OBC := LIMIT(0,diNrOfEM_IN_OBC,Constants_Energy.diMaxNumberOfElectricMeters);
			
(*------------------------------------------------------------------Power Data----------------------------------------------------------------------------*)

IF NOT bPowerDataInvers THEN
	fbOBC.lrCounterEnergyT1_Consumption := Lynus_Standards.GVL_Energy.stDataElectricMeters[diNrOfEM_IN_OBC].lrCounterEnergyT1_Production * 1000;
	fbOBC.lrCounterEnergyT2_Consumption := Lynus_Standards.GVL_Energy.stDataElectricMeters[diNrOfEM_IN_OBC].lrCounterEnergyT2_Production * 1000;
	fbOBC.lrCounterEnergyT1_Production := Lynus_Standards.GVL_Energy.stDataElectricMeters[diNrOfEM_IN_OBC].lrCounterEnergyT1_Consumption * 1000;
	fbOBC.lrCounterEnergyT2_Production := Lynus_Standards.GVL_Energy.stDataElectricMeters[diNrOfEM_IN_OBC].lrCounterEnergyT1_Consumption * 1000;
	fbOBC.lrTotalCounterEnergy_Consumption := Lynus_Standards.GVL_Energy.stDataElectricMeters[diNrOfEM_IN_OBC].lrTotalCounterEnergy_Production * 1000;
	fbOBC.lrTotalCounterEnergy_Production := Lynus_Standards.GVL_Energy.stDataElectricMeters[diNrOfEM_IN_OBC].lrTotalCounterEnergy_Consumption * 1000;
		fbOBC.lrPowerOBC := (Lynus_Standards.GVL_Energy.stDataElectricMeters[diNrOfEM_IN_OBC].lrPower * 1000) * - 1;
ELSE
	fbOBC.lrCounterEnergyT1_Consumption := Lynus_Standards.GVL_Energy.stDataElectricMeters[diNrOfEM_IN_OBC].lrCounterEnergyT1_Consumption * 1000;
	fbOBC.lrCounterEnergyT2_Consumption := Lynus_Standards.GVL_Energy.stDataElectricMeters[diNrOfEM_IN_OBC].lrCounterEnergyT2_Consumption * 1000;
	fbOBC.lrCounterEnergyT1_Production := Lynus_Standards.GVL_Energy.stDataElectricMeters[diNrOfEM_IN_OBC].lrCounterEnergyT1_Production * 1000;
	fbOBC.lrCounterEnergyT2_Production := Lynus_Standards.GVL_Energy.stDataElectricMeters[diNrOfEM_IN_OBC].lrCounterEnergyT2_Production * 1000;
	fbOBC.lrTotalCounterEnergy_Consumption := Lynus_Standards.GVL_Energy.stDataElectricMeters[diNrOfEM_IN_OBC].lrTotalCounterEnergy_Consumption * 1000;
	fbOBC.lrTotalCounterEnergy_Production := Lynus_Standards.GVL_Energy.stDataElectricMeters[diNrOfEM_IN_OBC].lrTotalCounterEnergy_Production * 1000;
		fbOBC.lrPowerOBC := Lynus_Standards.GVL_Energy.stDataElectricMeters[diNrOfEM_IN_OBC].lrPower * 1000;
END_IF

(*-------------------------------------------------------------Calcualte the number of OBC---------------------------------------------------------------*)

fbNumberDevice(
	diActualNumberOfDevices:= Lynus_Standards.GVL_Energy.stNumberOfDevices.diNumberOfOBC, 
	diMaxNumberOfDevices:= Constants_Energy.diMaxNumberOfOtherBigConsumers, 
	udiCounterOnlineChange:= TwinCAT_SystemInfoVarList._AppInfo.OnlineChangeCnt, 
	bNumberIsCalculatet=> , 
	bFPNumberIsCalculatet=> , 
	bOnlineChange=> , 
	diNumberForThisDevice=> diNrOfOBC_OUT, 
	diNumberOfTotalDevices=> );

//Write new Numer on GVL
IF fbNumberDevice.bFPNumberIsCalculatet THEN
	Lynus_Standards.GVL_Energy.stNumberOfDevices.diNumberOfOBC := fbNumberDevice.diNumberOfTotalDevices;	
END_IF 

//Delete old Number on GVL
IF fbNumberDevice.bOnlineChange THEN 
	Lynus_Standards.GVL_Energy.stNumberOfDevices.diNumberOfOBC := diNrOfOBC_OUT;	
		iStateGVLData := 1; 
END_IF

(*-------------------------------------------------------------Service from Backend is ready and check the connection to backen for dissabel/enable Function---------------------------------------------------------------*)

//Try to reset the variable for connection on the GVL. When all is normal then the Lynus Mqtt connection function set this variable to true in the next cycle
//When we have no connection to the backend then after Lynus_Standards.Constants_General.tTimeDissableLynusFunctions days the Function is dissabled with all of his functionalities
timResetConnectionOnGVL(IN:= NOT timResetConnectionOnGVL.Q, PT:= T#1H, Q=> , ET=> );
	IF timResetConnectionOnGVL.Q THEN Lynus_Standards.GVL_Communicator.bStateConnectionToEnableFunctions := FALSE; END_IF
		IF NOT Lynus_Standards.GVL_Communicator.bStateConnectionToEnableFunctions THEN timDissableFunctions.IN := TRUE; ELSE timDissableFunctions.IN := FALSE; END_IF  
			timDissableFunctions(IN:= , PT:= Lynus_Standards.Constants_General.tTimeDissableLynusFunctions, Q=> , ET=> );

(*------------------------------------------------------------------Error----------------------------------------------------------------------------*)

IF timDissableFunctions.Q THEN fbOBC.bWarning := TRUE; fbOBC.iWarningCode := 0; ELSE fbOBC.bWarning := FALSE; END_IF 
	IF Lynus_Standards.GVL_Energy.stNumberOfDevices.diNumberOfOBC > Constants_Energy.diMaxNumberOfOtherBigConsumers THEN 
		fbOBC.bError := TRUE;
			fbOBC.iErrorCode := 1; 
	ELSE 
		fbOBC.bError := FALSE; 
			fbOBC.iErrorCode := 0;
	END_IF 	
	
(*------------------------------------------------------------------Logic----------------------------------------------------------------------------*)
	
//Calcualte the total SOC if we have more then 1 battery in our system
diNumberOfActiveBatterys := 0;
	dwSumSOC := 0;
		FOR liLPBatteryData := 1 TO Constants_Energy.diMaxNumberOfBatterys BY 1 DO
			IF Lynus_Standards.GVL_Energy.stDataOfBatterys[diNrOfEMS_IN,liLPBatteryData].bEnabled THEN diNumberOfActiveBatterys := diNumberOfActiveBatterys + 1; END_IF
				dwSumSOC := dwSumSOC + Lynus_Standards.GVL_Energy.stDataOfBatterys[diNrOfEMS_IN,liLPBatteryData].dwSOC;
		END_FOR
	
IF diNumberOfActiveBatterys > 0 THEN
	fbOBC.dwBatterySOC := DINT_TO_DWORD(DWORD_TO_DINT(dwSumSOC) / diNumberOfActiveBatterys);
ELSE
	fbOBC.dwBatterySOC := 100;	//When we have no battery in the ems system
END_IF

//Check if one or more Batterysystems or batteryinverter make island mode
diNumberOfBatteryInverterInEPO := 0;
	FOR liLPInEPO := 1 TO Constants_Energy.diMaxNumberOfBatteryInverters BY 1 DO
		IF Lynus_Standards.GVL_Energy.stDataOfBatteryInverters[diNrOfEMS_IN,liLPInEPO].bWorkOnIslandMode THEN fbOBC.bEPOIsActive := TRUE; diNumberOfBatteryInverterInEPO := diNumberOfBatteryInverterInEPO + 1; END_IF
	END_FOR 
		IF diNumberOfBatteryInverterInEPO <= 0 THEN fbOBC.bEPOIsActive := FALSE; END_IF

//Digital input for external lock signal
fbDIExternalLock(bInvers:= FALSE, bSignal=> );

//Functionblock OBC
fbOBC(
	bEnable:= bEnable AND NOT timDissableFunctions.Q,
	bError:= , 
	bEPOIsActive:= , 
	bExternalLock:= fbDIExternalLock.bSignal, 
	bWriteWithDelay:= TRUE, 
	iErrorCode:= , 
	iWarningCode:= , 
	dwBatterySOC:= , 
	lrTotalCounterEnergy_Consumption:= , 
	lrTotalCounterEnergy_Production:= , 
	lrCounterEnergyT1_Consumption:= , 
	lrCounterEnergyT2_Consumption:= , 
	lrCounterEnergyT1_Production:= , 
	lrCounterEnergyT2_Production:= , 
	lrPowerOBC:= , 
	rTargetPower:= Lynus_Standards.GVL_Energy.stDataOtherBigConsumers[diNrOfEMS_IN,diNrOfOBC_OUT].rTargetPowerEMS, 
	tTimDelayOutput:= T#5S, 
	stSetupOBC:= stSetupOBC, 
	stDataOBCOut=> , 
	stDataOBCOutDelay=> stDataOBC);
						
(*-------------------------------------------------------------------------Output----------------------------------------------------------------------*)
	
IF bNoLinear THEN 
	fbInterpolation.rXInputValue := (stSetupOBC.rMaxPower * fbOBC.stDataOBCOut.rTargetPower) / 100; 
		fbInterpolation.arrYIntermediateValues[1] := 10;
			fbInterpolation.arrYIntermediateValues[2] := 20;
				fbInterpolation.arrYIntermediateValues[3] := 30;
					fbInterpolation.arrYIntermediateValues[4] := 40;
						fbInterpolation.arrYIntermediateValues[5] := 50;
	fbInterpolation.arrYIntermediateValues[6] := 60;
		fbInterpolation.arrYIntermediateValues[7] := 70;
			fbInterpolation.arrYIntermediateValues[8] := 80;
				fbInterpolation.arrYIntermediateValues[9] := 90;
					fbInterpolation.arrYIntermediateValues[10] := 100;
	fbInterpolation(rXInputValue:=, arrXIntermediateValues:= arrTableOfInterpolationPoints, arrYIntermediateValues:=, rYOutputValue=> );
END_IF

IF bNoLinear THEN 
	fbAOOBC.rSignal := fbInterpolation.rYOutputValue;
	//Target Power, to use this on a external Function
	rTargetPowerForExtFunc := fbInterpolation.rYOutputValue;
ELSE
	fbAOOBC.rSignal := fbOBC.stDataOBCOut.rTargetPower;
	//Target Power, to use this on a external Function
	rTargetPowerForExtFunc := fbOBC.stDataOBCOut.rTargetPower;
END_IF

fbAOOBC(
	rYMinTerminalValue:= 0, 
	rXMinInputSignal:= 0, 
	rYMaxTerminalValue:= 32767, 
	rXMaxInputSignal:= 100, 
	rSignal:= , 
	usiState=> );

(*-----------------------------------------------------------Handle data to Global structure for the other big consumers-----------------------------------------------------------------*)

//Delte al old Data on GVL after a online change or change on the variable diNrOfEMS_IDOD
IF diNrOfEMS_IN <> diNrOfEMS_IN_CP AND iStateGVLData = 0 THEN iStateGVLData := 10; END_IF 

CASE iStateGVLData OF
	
	0://Init Step
		byWaitInStep := 0;
			diCounterForGVL := 1;
	
	1://Wait for 4 Steps before clean al Data on GVL
		byWaitInStep := byWaitInStep + 1;
			IF byWaitInStep >= 4 AND fbNumberDevice.bNumberIsCalculatet THEN iStateGVLData := 2; END_IF
				//To much Devices, back to the Init step
				IF byWaitInStep >= 4 AND NOT fbNumberDevice.bNumberIsCalculatet THEN iStateGVLData := 0; END_IF	
			
	2://Clear all Data in GVL
		FOR diLPForGVL := 1 TO Constants_Energy.diMaxNumberOfEMS BY 1 DO 
			Lynus_Standards.GVL_Energy.stDataOtherBigConsumers[diLPForGVL,diCounterForGVL].bEnabled := FALSE;
				Lynus_Standards.GVL_Energy.stDataOtherBigConsumers[diLPForGVL,diCounterForGVL].bIsControllable := FALSE;
					Lynus_Standards.GVL_Energy.stDataOtherBigConsumers[diLPForGVL,diCounterForGVL].byPriority := 0;
						Lynus_Standards.GVL_Energy.stDataOtherBigConsumers[diLPForGVL,diCounterForGVL].byErrorWarning := 0;
							Lynus_Standards.GVL_Energy.stDataOtherBigConsumers[diLPForGVL,diCounterForGVL].lrPower := 0;
								Lynus_Standards.GVL_Energy.stDataOtherBigConsumers[diLPForGVL,diCounterForGVL].lrPowerConsumption := 0;
									Lynus_Standards.GVL_Energy.stDataOtherBigConsumers[diLPForGVL,diCounterForGVL].lrPowerProduction := 0;
										Lynus_Standards.GVL_Energy.stDataOtherBigConsumers[diLPForGVL,diCounterForGVL].rMaxPower := 0;
											//Set also the target value from ems back here to 0 and not in EMS function because EMS is in Standy when we have a online change (Problem when we delete a ems function and make a online change)
											Lynus_Standards.GVL_Energy.stDataOtherBigConsumers[diLPForGVL,diCounterForGVL].rTargetPowerEMS := 0;
		END_FOR
			diCounterForGVL := diCounterForGVL + 1;
				diCounterForGVL := LIMIT(0,diCounterForGVL,Constants_Energy.diMaxNumberOfOtherBigConsumers);
					//Back to the init step
					IF diCounterForGVL >= Constants_Energy.diMaxNumberOfOtherBigConsumers THEN iStateGVLData := 0; END_IF

	10://Clear old Data on GVL 	
		Lynus_Standards.GVL_Energy.stDataOtherBigConsumers[diNrOfEMS_IN_CP,diNrOfOBC_OUT].bEnabled := FALSE;
			Lynus_Standards.GVL_Energy.stDataOtherBigConsumers[diNrOfEMS_IN_CP,diNrOfOBC_OUT].bIsControllable := FALSE;
				Lynus_Standards.GVL_Energy.stDataOtherBigConsumers[diNrOfEMS_IN_CP,diNrOfOBC_OUT].byPriority := 0;
					Lynus_Standards.GVL_Energy.stDataOtherBigConsumers[diNrOfEMS_IN_CP,diNrOfOBC_OUT].byErrorWarning := 0;
						Lynus_Standards.GVL_Energy.stDataOtherBigConsumers[diNrOfEMS_IN_CP,diNrOfOBC_OUT].lrPower := 0;
							Lynus_Standards.GVL_Energy.stDataOtherBigConsumers[diNrOfEMS_IN_CP,diNrOfOBC_OUT].lrPowerConsumption := 0;
								Lynus_Standards.GVL_Energy.stDataOtherBigConsumers[diNrOfEMS_IN_CP,diNrOfOBC_OUT].lrPowerProduction := 0;
									Lynus_Standards.GVL_Energy.stDataOtherBigConsumers[diNrOfEMS_IN_CP,diNrOfOBC_OUT].rMaxPower := 0;
	
		diNrOfEMS_IN_CP := diNrOfEMS_IN;
			//Back to the init step
			iStateGVLData := 0;

END_CASE 	 

IF diNrOfOBC_OUT > 0 AND fbNumberDevice.bNumberIsCalculatet AND diNrOfEMS_IN > 0 THEN
	Lynus_Standards.GVL_Energy.stDataOtherBigConsumers[diNrOfEMS_IN,diNrOfOBC_OUT].bEnabled := fbOBC.stDataOBCOut.bEnabled;
		Lynus_Standards.GVL_Energy.stDataOtherBigConsumers[diNrOfEMS_IN,diNrOfOBC_OUT].bIsControllable := TRUE;
			Lynus_Standards.GVL_Energy.stDataOtherBigConsumers[diNrOfEMS_IN,diNrOfOBC_OUT].byPriority := fbOBC.stDataOBCOut.byPriority;
				Lynus_Standards.GVL_Energy.stDataOtherBigConsumers[diNrOfEMS_IN,diNrOfOBC_OUT].byErrorWarning := fbOBC.stDataOBCOut.byErrorWarning;
					Lynus_Standards.GVL_Energy.stDataOtherBigConsumers[diNrOfEMS_IN,diNrOfOBC_OUT].lrPower := fbOBC.stDataOBCOut.lrPower;
						Lynus_Standards.GVL_Energy.stDataOtherBigConsumers[diNrOfEMS_IN,diNrOfOBC_OUT].lrPowerConsumption := fbOBC.stDataOBCOut.lrPowerConsumption;
							Lynus_Standards.GVL_Energy.stDataOtherBigConsumers[diNrOfEMS_IN,diNrOfOBC_OUT].lrPowerProduction := fbOBC.stDataOBCOut.lrPowerProduction;
								Lynus_Standards.GVL_Energy.stDataOtherBigConsumers[diNrOfEMS_IN,diNrOfOBC_OUT].rMaxPower := fbOBC.stDataOBCOut.rMaxPower;
END_IF

(*----------------------------------------------------------Save persistent data----------------------------------------------------------------*)

arrPD[1](lrValue:= BOOL_TO_LREAL(bEnable), bEventBasedActive=> );
arrPD[2](lrValue:= BOOL_TO_LREAL(bPowerDataInvers), bEventBasedActive=> );
arrPD[3](lrValue:= DINT_TO_LREAL(diNrOfEMS_IN), bEventBasedActive=> );
arrPD[4](lrValue:= DINT_TO_LREAL(diNrOfEM_IN_OBC), bEventBasedActive=> );
arrPD[5](lrValue:= DINT_TO_LREAL(diNrOfEMS_IN_CP), bEventBasedActive=> );
arrPD[6](lrValue:= BOOL_TO_LREAL(stSetupOBC.bManualyOn), bEventBasedActive=> );
arrPD[7](lrValue:= BOOL_TO_LREAL(stSetupOBC.bOnEmergPowerOff), bEventBasedActive=> );
arrPD[8](lrValue:= BYTE_TO_LREAL(stSetupOBC.byDisableSOC), bEventBasedActive=> );
arrPD[9](lrValue:= BYTE_TO_LREAL(stSetupOBC.byEnableSOC), bEventBasedActive=> );
arrPD[10](lrValue:= BYTE_TO_LREAL(stSetupOBC.byManualyTargetPower), bEventBasedActive=> );
arrPD[11](lrValue:= BYTE_TO_LREAL(stSetupOBC.byPriority), bEventBasedActive=> );
arrPD[12](lrValue:= REAL_TO_LREAL(stSetupOBC.rMaxPower), bEventBasedActive=> );
arrPD[13](lrValue:= BOOL_TO_LREAL(bNoLinear), bEventBasedActive=> );
arrPD[14](lrValue:= REAL_TO_LREAL(arrTableOfInterpolationPoints[1]), bEventBasedActive=> );
arrPD[15](lrValue:= REAL_TO_LREAL(arrTableOfInterpolationPoints[2]), bEventBasedActive=> );
arrPD[16](lrValue:= REAL_TO_LREAL(arrTableOfInterpolationPoints[3]), bEventBasedActive=> );
arrPD[17](lrValue:= REAL_TO_LREAL(arrTableOfInterpolationPoints[4]), bEventBasedActive=> );
arrPD[18](lrValue:= REAL_TO_LREAL(arrTableOfInterpolationPoints[5]), bEventBasedActive=> );
arrPD[19](lrValue:= REAL_TO_LREAL(arrTableOfInterpolationPoints[6]), bEventBasedActive=> );
arrPD[20](lrValue:= REAL_TO_LREAL(arrTableOfInterpolationPoints[7]), bEventBasedActive=> );
arrPD[21](lrValue:= REAL_TO_LREAL(arrTableOfInterpolationPoints[8]), bEventBasedActive=> );
arrPD[22](lrValue:= REAL_TO_LREAL(arrTableOfInterpolationPoints[9]), bEventBasedActive=> );
arrPD[23](lrValue:= REAL_TO_LREAL(arrTableOfInterpolationPoints[10]), bEventBasedActive=> );

END_FUNCTION_BLOCK

// ---- FBs/Other Big Consumer/OnOff/FB_OBC_OnOff.TcPOU
FUNCTION_BLOCK FB_OBC_OnOff
VAR_INPUT PERSISTENT
	bEnable									: BOOL;												//{#lynus.ag#()} //Enable the Fuctionblock and his logic
	bPowerDataInvers						: BOOL;												//With True its possible to invert all received power data from the electric meter
	diNrOfEMS_IN							: DINT;												//Number of EMS what control this Device.
	diNrOfEM_IN_OBC							: DINT;												//Number of the electric meter for incoming power data. (Power Data for this Device)
	stSetupOBC								: ST_Setup_OBC;										//{#lynus.ag#()} //Setup other big consumer
END_VAR
VAR_INPUT
END_VAR
VAR_OUTPUT
	stDataOBC								: ST_OBC_Output;									//{#lynus.ag#()} //Output Data other big consumer
	diNrOfOBC_OUT							: DINT;												//Active Number from the other big consumer for using on other functions
	rTargetPowerForExtFunc					: REAL;												//Target Power from 0% to +100% to use on a external Function
END_VAR
VAR
	{attribute 'hide'}
	fbOBC									: FB_BigConsumer;									//Function for other big consumer
	{attribute 'hide'}
	fbNumberDevice							: FB_NumberOfDevice;								//Function block to calcualte the number of the Device
	fbDIExternalLock						: FB_XL1XXX_DI;										//Digital Input from external loock signal
	fbDOOnOffOBC							: FB_XL2XXX_DO;										//Digital Output to swtich on and off the OBC
	{attribute 'hide'}
	timDissableFunctions					: TON;												//Timer to dissable the Function after Lynus_Standards.Constants_General.tTimeDissableLynusFunctions Days without connection to the Lynus Cloud
	{attribute 'hide'}
	timResetConnectionOnGVL					: TON;												//Timer to try reset the connection Flag on the GVL. (When somebody delete the Connection Function and make only a onlinechange)
	{attribute 'hide'}
	arrPD									: ARRAY[1..12] OF FB_PersistentData_Number;			//Function to save persistent data 
	{attribute 'hide'}
	byWaitInStep							: BYTE;												//Wait in Step before start to clean data on PLC
	{attribute 'hide'}
	iStateGVLData							: INT;												//State machine to handle the data on the GVL
	{attribute 'hide'}
	diNumberOfActiveBatterys				: DINT;												//Number of active batterys
	{attribute 'hide'}
	diNumberOfBatteryInverterInEPO			: DINT;												//Number of battery inverters that work in Emergency Power operation 
	{attribute 'hide'}
	diCounterForGVL							: DINT;												//Counter to clean old data on GVL
	{attribute 'hide'}
	diLPForGVL								: DINT;												//Loop to clean old data on GVL
	{attribute 'hide'}
	dwSumSOC								: DWORD;											//Sum of the SOC from all batterys
	{attribute 'hide'}
	liLPBatteryData							: LINT;												//Loop to check some data from batterys
	{attribute 'hide'}
	liLPInEPO								: LINT;												//Loop to check if 1 or more battery inverters build a island grid	
END_VAR
VAR PERSISTENT
	{attribute 'conditionalshow'}
	diNrOfEMS_IN_CP							: DINT;												//Number of EMS what control this Device to compare with the original
END_VAR

//Creator : Kai Ebensperger
//Company : Lynus AG
//Date : 19.05.2021
//Version : 1.0.0.0

//With this function block its possible to control a other big consumer with the plc
//The output signal to control the big consumer is a digital output signal
//Also the Power Data can by displayed with this functionblock

//NOTE for diNr.....Designation => 
//_IN = Here Data come in from other Functions or go out to other functions about the GVL
//_OUT = Here Data go out to other functions about the GVL

(*------------------------------------------------------------Limits----------------------------------------------------------------------------------*)

diNrOfEMS_IN := LIMIT(0,diNrOfEMS_IN,Constants_Energy.diMaxNumberOfEMS);
	diNrOfEM_IN_OBC := LIMIT(0,diNrOfEM_IN_OBC,Constants_Energy.diMaxNumberOfElectricMeters);
			
(*------------------------------------------------------------------Power Data----------------------------------------------------------------------------*)

IF NOT bPowerDataInvers THEN
	fbOBC.lrCounterEnergyT1_Consumption := Lynus_Standards.GVL_Energy.stDataElectricMeters[diNrOfEM_IN_OBC].lrCounterEnergyT1_Production * 1000;
	fbOBC.lrCounterEnergyT2_Consumption := Lynus_Standards.GVL_Energy.stDataElectricMeters[diNrOfEM_IN_OBC].lrCounterEnergyT2_Production * 1000;
	fbOBC.lrCounterEnergyT1_Production := Lynus_Standards.GVL_Energy.stDataElectricMeters[diNrOfEM_IN_OBC].lrCounterEnergyT1_Consumption * 1000;
	fbOBC.lrCounterEnergyT2_Production := Lynus_Standards.GVL_Energy.stDataElectricMeters[diNrOfEM_IN_OBC].lrCounterEnergyT1_Consumption * 1000;
	fbOBC.lrTotalCounterEnergy_Consumption := Lynus_Standards.GVL_Energy.stDataElectricMeters[diNrOfEM_IN_OBC].lrTotalCounterEnergy_Production * 1000;
	fbOBC.lrTotalCounterEnergy_Production := Lynus_Standards.GVL_Energy.stDataElectricMeters[diNrOfEM_IN_OBC].lrTotalCounterEnergy_Consumption * 1000;
		fbOBC.lrPowerOBC := (Lynus_Standards.GVL_Energy.stDataElectricMeters[diNrOfEM_IN_OBC].lrPower * 1000) * - 1;
ELSE
	fbOBC.lrCounterEnergyT1_Consumption := Lynus_Standards.GVL_Energy.stDataElectricMeters[diNrOfEM_IN_OBC].lrCounterEnergyT1_Consumption * 1000;
	fbOBC.lrCounterEnergyT2_Consumption := Lynus_Standards.GVL_Energy.stDataElectricMeters[diNrOfEM_IN_OBC].lrCounterEnergyT2_Consumption * 1000;
	fbOBC.lrCounterEnergyT1_Production := Lynus_Standards.GVL_Energy.stDataElectricMeters[diNrOfEM_IN_OBC].lrCounterEnergyT1_Production * 1000;
	fbOBC.lrCounterEnergyT2_Production := Lynus_Standards.GVL_Energy.stDataElectricMeters[diNrOfEM_IN_OBC].lrCounterEnergyT2_Production * 1000;
	fbOBC.lrTotalCounterEnergy_Consumption := Lynus_Standards.GVL_Energy.stDataElectricMeters[diNrOfEM_IN_OBC].lrTotalCounterEnergy_Consumption * 1000;
	fbOBC.lrTotalCounterEnergy_Production := Lynus_Standards.GVL_Energy.stDataElectricMeters[diNrOfEM_IN_OBC].lrTotalCounterEnergy_Production * 1000;
		fbOBC.lrPowerOBC := Lynus_Standards.GVL_Energy.stDataElectricMeters[diNrOfEM_IN_OBC].lrPower * 1000;
END_IF

(*-------------------------------------------------------------Calcualte the number of OBC---------------------------------------------------------------*)

fbNumberDevice(
	diActualNumberOfDevices:= Lynus_Standards.GVL_Energy.stNumberOfDevices.diNumberOfOBC, 
	diMaxNumberOfDevices:= Constants_Energy.diMaxNumberOfOtherBigConsumers, 
	udiCounterOnlineChange:= TwinCAT_SystemInfoVarList._AppInfo.OnlineChangeCnt, 
	bNumberIsCalculatet=> , 
	bFPNumberIsCalculatet=> , 
	bOnlineChange=> , 
	diNumberForThisDevice=> diNrOfOBC_OUT, 
	diNumberOfTotalDevices=> );

//Write new Numer on GVL
IF fbNumberDevice.bFPNumberIsCalculatet THEN
	Lynus_Standards.GVL_Energy.stNumberOfDevices.diNumberOfOBC := fbNumberDevice.diNumberOfTotalDevices;	
END_IF 

//Delete old Number on GVL
IF fbNumberDevice.bOnlineChange THEN 
	Lynus_Standards.GVL_Energy.stNumberOfDevices.diNumberOfOBC := diNrOfOBC_OUT;	
		iStateGVLData := 1; 
END_IF

(*-------------------------------------------------------------Service from Backend is ready and check the connection to backen for dissabel/enable Function---------------------------------------------------------------*)

//Try to reset the variable for connection on the GVL. When all is normal then the Lynus Mqtt connection function set this variable to true in the next cycle
//When we have no connection to the backend then after Lynus_Standards.Constants_General.tTimeDissableLynusFunctions days the Function is dissabled with all of his functionalities
timResetConnectionOnGVL(IN:= NOT timResetConnectionOnGVL.Q, PT:= T#1H, Q=> , ET=> );
	IF timResetConnectionOnGVL.Q THEN Lynus_Standards.GVL_Communicator.bStateConnectionToEnableFunctions := FALSE; END_IF
		IF NOT Lynus_Standards.GVL_Communicator.bStateConnectionToEnableFunctions THEN timDissableFunctions.IN := TRUE; ELSE timDissableFunctions.IN := FALSE; END_IF  
			timDissableFunctions(IN:= , PT:= Lynus_Standards.Constants_General.tTimeDissableLynusFunctions, Q=> , ET=> );

(*------------------------------------------------------------------Error----------------------------------------------------------------------------*)

IF timDissableFunctions.Q THEN fbOBC.bWarning := TRUE; fbOBC.iWarningCode := 0; ELSE fbOBC.bWarning := FALSE; END_IF 
	IF Lynus_Standards.GVL_Energy.stNumberOfDevices.diNumberOfOBC > Constants_Energy.diMaxNumberOfOtherBigConsumers THEN 
		fbOBC.bError := TRUE;
			fbOBC.iErrorCode := 1; 
	ELSE 
		fbOBC.bError := FALSE; 
			fbOBC.iErrorCode := 0;
	END_IF 	
	
(*------------------------------------------------------------------Logic----------------------------------------------------------------------------*)
	
//Calcualte the total SOC if we have more then 1 battery in our system
diNumberOfActiveBatterys := 0;
	dwSumSOC := 0;
		FOR liLPBatteryData := 1 TO Constants_Energy.diMaxNumberOfBatterys BY 1 DO
			IF Lynus_Standards.GVL_Energy.stDataOfBatterys[diNrOfEMS_IN,liLPBatteryData].bEnabled THEN diNumberOfActiveBatterys := diNumberOfActiveBatterys + 1; END_IF
				dwSumSOC := dwSumSOC + Lynus_Standards.GVL_Energy.stDataOfBatterys[diNrOfEMS_IN,liLPBatteryData].dwSOC;
		END_FOR
	
IF diNumberOfActiveBatterys > 0 THEN
	fbOBC.dwBatterySOC := DINT_TO_DWORD(DWORD_TO_DINT(dwSumSOC) / diNumberOfActiveBatterys);
ELSE
	fbOBC.dwBatterySOC := 100;	//When we have no battery in the ems system
END_IF

//Check if one or more Batterysystems or batteryinverter make island mode
diNumberOfBatteryInverterInEPO := 0;
	FOR liLPInEPO := 1 TO Constants_Energy.diMaxNumberOfBatteryInverters BY 1 DO
		IF Lynus_Standards.GVL_Energy.stDataOfBatteryInverters[diNrOfEMS_IN,liLPInEPO].bWorkOnIslandMode THEN fbOBC.bEPOIsActive := TRUE; diNumberOfBatteryInverterInEPO := diNumberOfBatteryInverterInEPO + 1; END_IF
	END_FOR 
		IF diNumberOfBatteryInverterInEPO <= 0 THEN fbOBC.bEPOIsActive := FALSE; END_IF

//Digital input for external lock signal
fbDIExternalLock(bInvers:= FALSE, bSignal=> );

//Functionblock OBC
fbOBC.stSetupOBC.bManualyOn := stSetupOBC.bManualyOn;
	IF fbOBC.stSetupOBC.bManualyOn THEN fbOBC.stSetupOBC.byManualyTargetPower := 100; ELSE fbOBC.stSetupOBC.byManualyTargetPower := 0; END_IF
		fbOBC.stSetupOBC.bOnEmergPowerOff := stSetupOBC.bOnEmergPowerOff;
			fbOBC.stSetupOBC.byDisableSOC := stSetupOBC.byDisableSOC;
				fbOBC.stSetupOBC.byEnableSOC := stSetupOBC.byEnableSOC;
					fbOBC.stSetupOBC.byPriority := stSetupOBC.byPriority;
						fbOBC.stSetupOBC.rMaxPower := stSetupOBC.rMaxPower;	

fbOBC(
	bEnable:= bEnable AND NOT timDissableFunctions.Q,
	bError:= , 
	bEPOIsActive:= , 
	bExternalLock:= fbDIExternalLock.bSignal, 
	bWriteWithDelay:= TRUE, 
	iErrorCode:= , 
	iWarningCode:= , 
	dwBatterySOC:= , 
	lrTotalCounterEnergy_Consumption:= , 
	lrTotalCounterEnergy_Production:= , 
	lrCounterEnergyT1_Consumption:= , 
	lrCounterEnergyT2_Consumption:= , 
	lrCounterEnergyT1_Production:= , 
	lrCounterEnergyT2_Production:= , 
	lrPowerOBC:= , 
	rTargetPower:= Lynus_Standards.GVL_Energy.stDataOtherBigConsumers[diNrOfEMS_IN,diNrOfOBC_OUT].rTargetPowerEMS, 
	tTimDelayOutput:= T#5S, 
	stSetupOBC:= , 
	stDataOBCOut=> , 
	stDataOBCOutDelay=> stDataOBC);											

//Target Power, to use this on a external Function
rTargetPowerForExtFunc := fbOBC.stDataOBCOut.rTargetPower;
	
(*-------------------------------------------------------------------------Output----------------------------------------------------------------------*)
	
fbDOOnOffOBC(bInvers:= FALSE, bSignal:= fbOBC.stDataOBCOut.bOutputOnOff);

(*-----------------------------------------------------------Handle data to Global structure for the other big consumers-----------------------------------------------------------------*)

//Delte al old Data on GVL after a online change or change on the variable diNrOfEMS_IDOD
IF diNrOfEM_IN_OBC <> diNrOfEMS_IN_CP AND iStateGVLData = 0 THEN iStateGVLData := 10; END_IF 

CASE iStateGVLData OF
	
	0://Init Step
		byWaitInStep := 0;
			diCounterForGVL := 1;
	
	1://Wait for 4 Steps before clean al Data on GVL
		byWaitInStep := byWaitInStep + 1;
			IF byWaitInStep >= 4 AND fbNumberDevice.bNumberIsCalculatet THEN iStateGVLData := 2; END_IF
				//To much Devices, back to the Init step
				IF byWaitInStep >= 4 AND NOT fbNumberDevice.bNumberIsCalculatet THEN iStateGVLData := 0; END_IF	
			
	2://Clear all Data in GVL
		FOR diLPForGVL := 1 TO Constants_Energy.diMaxNumberOfEMS BY 1 DO 
			Lynus_Standards.GVL_Energy.stDataOtherBigConsumers[diLPForGVL,diCounterForGVL].bEnabled := FALSE;
				Lynus_Standards.GVL_Energy.stDataOtherBigConsumers[diLPForGVL,diCounterForGVL].bIsControllable := FALSE;
					Lynus_Standards.GVL_Energy.stDataOtherBigConsumers[diLPForGVL,diCounterForGVL].byPriority := 0;
						Lynus_Standards.GVL_Energy.stDataOtherBigConsumers[diLPForGVL,diCounterForGVL].byErrorWarning := 0;
							Lynus_Standards.GVL_Energy.stDataOtherBigConsumers[diLPForGVL,diCounterForGVL].lrPower := 0;
								Lynus_Standards.GVL_Energy.stDataOtherBigConsumers[diLPForGVL,diCounterForGVL].lrPowerConsumption := 0;
									Lynus_Standards.GVL_Energy.stDataOtherBigConsumers[diLPForGVL,diCounterForGVL].lrPowerProduction := 0;
										Lynus_Standards.GVL_Energy.stDataOtherBigConsumers[diLPForGVL,diCounterForGVL].rMaxPower := 0;
											//Set also the target value from ems back here to 0 and not in EMS function because EMS is in Standy when we have a online change (Problem when we delete a ems function and make a online change)
											Lynus_Standards.GVL_Energy.stDataOtherBigConsumers[diLPForGVL,diCounterForGVL].rTargetPowerEMS := 0;
		END_FOR
			diCounterForGVL := diCounterForGVL + 1;
				diCounterForGVL := LIMIT(0,diCounterForGVL,Constants_Energy.diMaxNumberOfOtherBigConsumers);
					//Back to the init step
					IF diCounterForGVL >= Constants_Energy.diMaxNumberOfOtherBigConsumers THEN iStateGVLData := 0; END_IF

	10://Clear old Data on GVL 	
		Lynus_Standards.GVL_Energy.stDataOtherBigConsumers[diNrOfEMS_IN_CP,diNrOfOBC_OUT].bEnabled := FALSE;
			Lynus_Standards.GVL_Energy.stDataOtherBigConsumers[diNrOfEMS_IN_CP,diNrOfOBC_OUT].bIsControllable := FALSE;
				Lynus_Standards.GVL_Energy.stDataOtherBigConsumers[diNrOfEMS_IN_CP,diNrOfOBC_OUT].byPriority := 0;
					Lynus_Standards.GVL_Energy.stDataOtherBigConsumers[diNrOfEMS_IN_CP,diNrOfOBC_OUT].byErrorWarning := 0;
						Lynus_Standards.GVL_Energy.stDataOtherBigConsumers[diNrOfEMS_IN_CP,diNrOfOBC_OUT].lrPower := 0;
							Lynus_Standards.GVL_Energy.stDataOtherBigConsumers[diNrOfEMS_IN_CP,diNrOfOBC_OUT].lrPowerConsumption := 0;
								Lynus_Standards.GVL_Energy.stDataOtherBigConsumers[diNrOfEMS_IN_CP,diNrOfOBC_OUT].lrPowerProduction := 0;
									Lynus_Standards.GVL_Energy.stDataOtherBigConsumers[diNrOfEMS_IN_CP,diNrOfOBC_OUT].rMaxPower := 0;
	
		diNrOfEMS_IN_CP := diNrOfEMS_IN;
			//Back to the init step
			iStateGVLData := 0;

END_CASE 	 

IF diNrOfOBC_OUT > 0 AND fbNumberDevice.bNumberIsCalculatet AND diNrOfEMS_IN > 0 THEN
	Lynus_Standards.GVL_Energy.stDataOtherBigConsumers[diNrOfEMS_IN,diNrOfOBC_OUT].bEnabled := fbOBC.stDataOBCOut.bEnabled;
		Lynus_Standards.GVL_Energy.stDataOtherBigConsumers[diNrOfEMS_IN,diNrOfOBC_OUT].bIsControllable := FALSE;
			Lynus_Standards.GVL_Energy.stDataOtherBigConsumers[diNrOfEMS_IN,diNrOfOBC_OUT].byPriority := fbOBC.stDataOBCOut.byPriority;
				Lynus_Standards.GVL_Energy.stDataOtherBigConsumers[diNrOfEMS_IN,diNrOfOBC_OUT].byErrorWarning := fbOBC.stDataOBCOut.byErrorWarning;
					Lynus_Standards.GVL_Energy.stDataOtherBigConsumers[diNrOfEMS_IN,diNrOfOBC_OUT].lrPower := fbOBC.stDataOBCOut.lrPower;
						Lynus_Standards.GVL_Energy.stDataOtherBigConsumers[diNrOfEMS_IN,diNrOfOBC_OUT].lrPowerConsumption := fbOBC.stDataOBCOut.lrPowerConsumption;
							Lynus_Standards.GVL_Energy.stDataOtherBigConsumers[diNrOfEMS_IN,diNrOfOBC_OUT].lrPowerProduction := fbOBC.stDataOBCOut.lrPowerProduction;
								Lynus_Standards.GVL_Energy.stDataOtherBigConsumers[diNrOfEMS_IN,diNrOfOBC_OUT].rMaxPower := fbOBC.stDataOBCOut.rMaxPower;
END_IF

(*----------------------------------------------------------Save persistent data----------------------------------------------------------------*)

arrPD[1](lrValue:= BOOL_TO_LREAL(bEnable), bEventBasedActive=> );
arrPD[2](lrValue:= BOOL_TO_LREAL(bPowerDataInvers), bEventBasedActive=> );
arrPD[3](lrValue:= DINT_TO_LREAL(diNrOfEMS_IN), bEventBasedActive=> );
arrPD[4](lrValue:= DINT_TO_LREAL(diNrOfEM_IN_OBC), bEventBasedActive=> );
arrPD[5](lrValue:= DINT_TO_LREAL(diNrOfEMS_IN_CP), bEventBasedActive=> );
arrPD[6](lrValue:= BOOL_TO_LREAL(stSetupOBC.bManualyOn), bEventBasedActive=> );
arrPD[7](lrValue:= BOOL_TO_LREAL(stSetupOBC.bOnEmergPowerOff), bEventBasedActive=> );
arrPD[8](lrValue:= BYTE_TO_LREAL(stSetupOBC.byDisableSOC), bEventBasedActive=> );
arrPD[9](lrValue:= BYTE_TO_LREAL(stSetupOBC.byEnableSOC), bEventBasedActive=> );
arrPD[10](lrValue:= BYTE_TO_LREAL(stSetupOBC.byManualyTargetPower), bEventBasedActive=> );
arrPD[11](lrValue:= BYTE_TO_LREAL(stSetupOBC.byPriority), bEventBasedActive=> );
arrPD[12](lrValue:= REAL_TO_LREAL(stSetupOBC.rMaxPower), bEventBasedActive=> );

END_FUNCTION_BLOCK

// ---- FBs/PV/FB_PV_Power.TcPOU
FUNCTION_BLOCK FB_PV_Power
VAR_INPUT PERSISTENT
	bEnable									: BOOL;													//Enable the Fuctionblock and his logic
	bPowerDataInvers						: BOOL;													//With True its possible to invert all received power data from the electric meter
	diNrOfEM_IN_PV							: DINT;													//Number of the electric meter for incoming power data. (Power Data for this Device)
END_VAR
VAR_INPUT
END_VAR
VAR_OUTPUT
	stDataPv								: ST_PV_Output;											//{#lynus.ag#()} //Output Data Pv System
	diNrOfPv_OUT							: DINT;													//Active Number from the Pv system for using on other functions
END_VAR
VAR
	{attribute 'hide'}
	fbPv									: FB_PV_Production;										//Function block for Pv system
	{attribute 'hide'}
	fbNumberDevice							: FB_NumberOfDevice;									//Function block to calcualte the number of the Device
	fbDIErrorPv								: FB_XL1XXX_DI;											//Digital Input Error Pv System
	{attribute 'hide'}
	timDissableFunctions					: TON;													//Timer to dissable the Function after Lynus_Standards.Constants_General.tTimeDissableLynusFunctions Days without connection to the Lynus Cloud
	{attribute 'hide'}
	timResetConnectionOnGVL					: TON;													//Timer to try reset the connection Flag on the GVL. (When somebody delete the Connection Function and make only a onlinechange)
	{attribute 'hide'}
	arrPD									: ARRAY[1..3] OF FB_PersistentData_Number;				//Function to save persistent data 
	{attribute 'hide'}
	byWaitInStep							: BYTE;													//Wait in Step before start to clean data on PLC
	{attribute 'hide'}
	iStateGVLData							: INT;													//State machine to handle the data on the GVL
	{attribute 'hide'}
	diCounterForGVL							: DINT;													//Counter to clean old data on GVL
END_VAR

//Creator : Kai Ebensperger
//Company : Lynus AG
//Date : 08.06.2021
//Version : 1.0.0.0

//With this function block its possible to show the power data from a pv system.
//This function block has no active communication to a pv system. Visualize only the received power data
//This function has a DI Signal for a external Error from the Pv system

//NOTE for diNr.....Designation => 
//_IN = Here Data come in from other Functions or go out to other functions about the GVL
//_OUT = Here Data go out to other functions about the GVL

(*------------------------------------------------------------Limits----------------------------------------------------------------------------------*)

diNrOfEM_IN_PV := LIMIT(0,diNrOfEM_IN_PV,Constants_Energy.diMaxNumberOfElectricMeters);	

(*------------------------------------------------------------------Power Data----------------------------------------------------------------------------*)

IF NOT bPowerDataInvers THEN
	fbPv.lrCounterEnergyT1_Consumption := Lynus_Standards.GVL_Energy.stDataElectricMeters[diNrOfEM_IN_PV].lrCounterEnergyT1_Production * 1000;
	fbPv.lrCounterEnergyT2_Consumption := Lynus_Standards.GVL_Energy.stDataElectricMeters[diNrOfEM_IN_PV].lrCounterEnergyT2_Production * 1000;
	fbPv.lrCounterEnergyT1_Production := Lynus_Standards.GVL_Energy.stDataElectricMeters[diNrOfEM_IN_PV].lrCounterEnergyT1_Consumption * 1000;
	fbPv.lrCounterEnergyT2_Production := Lynus_Standards.GVL_Energy.stDataElectricMeters[diNrOfEM_IN_PV].lrCounterEnergyT1_Consumption * 1000;
	fbPv.lrTotalCounterEnergy_Consumption := Lynus_Standards.GVL_Energy.stDataElectricMeters[diNrOfEM_IN_PV].lrTotalCounterEnergy_Production * 1000;
	fbPv.lrTotalCounterEnergy_Production := Lynus_Standards.GVL_Energy.stDataElectricMeters[diNrOfEM_IN_PV].lrTotalCounterEnergy_Consumption * 1000;
ELSE
	fbPv.lrCounterEnergyT1_Consumption := Lynus_Standards.GVL_Energy.stDataElectricMeters[diNrOfEM_IN_PV].lrCounterEnergyT1_Consumption * 1000;
	fbPv.lrCounterEnergyT2_Consumption := Lynus_Standards.GVL_Energy.stDataElectricMeters[diNrOfEM_IN_PV].lrCounterEnergyT2_Consumption * 1000;
	fbPv.lrCounterEnergyT1_Production := Lynus_Standards.GVL_Energy.stDataElectricMeters[diNrOfEM_IN_PV].lrCounterEnergyT1_Production * 1000;
	fbPv.lrCounterEnergyT2_Production := Lynus_Standards.GVL_Energy.stDataElectricMeters[diNrOfEM_IN_PV].lrCounterEnergyT2_Production * 1000;
	fbPv.lrTotalCounterEnergy_Consumption := Lynus_Standards.GVL_Energy.stDataElectricMeters[diNrOfEM_IN_PV].lrTotalCounterEnergy_Consumption * 1000;
	fbPv.lrTotalCounterEnergy_Production := Lynus_Standards.GVL_Energy.stDataElectricMeters[diNrOfEM_IN_PV].lrTotalCounterEnergy_Production * 1000;
		
END_IF	

(*-------------------------------------------------------------Calcualte the number of Pv System---------------------------------------------------------------*)

fbNumberDevice(
	diActualNumberOfDevices:= Lynus_Standards.GVL_Energy.stNumberOfDevices.diNumberOfPvSystems, 
	diMaxNumberOfDevices:= Constants_Energy.diMaxNumberOfPvSystems, 
	udiCounterOnlineChange:= TwinCAT_SystemInfoVarList._AppInfo.OnlineChangeCnt, 
	bNumberIsCalculatet=> , 
	bFPNumberIsCalculatet=> , 
	bOnlineChange=> , 
	diNumberForThisDevice=> diNrOfPv_OUT, 
	diNumberOfTotalDevices=> );

//Write new Numer on GVL
IF fbNumberDevice.bFPNumberIsCalculatet THEN
	Lynus_Standards.GVL_Energy.stNumberOfDevices.diNumberOfPvSystems := fbNumberDevice.diNumberOfTotalDevices;	
END_IF 

//Delete old Number on GVL
IF fbNumberDevice.bOnlineChange THEN 
	Lynus_Standards.GVL_Energy.stNumberOfDevices.diNumberOfPvSystems := diNrOfPv_OUT;	
		iStateGVLData := 1; 
END_IF	

(*-------------------------------------------------------------Service from Backend is ready and check the connection to backen for dissabel/enable Function---------------------------------------------------------------*)

//Try to reset the variable for connection on the GVL. When all is normal then the Lynus Mqtt connection function set this variable to true in the next cycle
//When we have no connection to the backend then after Lynus_Standards.Constants_General.tTimeDissableLynusFunctions days the Function is dissabled with all of his functionalities
timResetConnectionOnGVL(IN:= NOT timResetConnectionOnGVL.Q, PT:= T#1H, Q=> , ET=> );
	IF timResetConnectionOnGVL.Q THEN Lynus_Standards.GVL_Communicator.bStateConnectionToEnableFunctions := FALSE; END_IF
		IF NOT Lynus_Standards.GVL_Communicator.bStateConnectionToEnableFunctions THEN timDissableFunctions.IN := TRUE; ELSE timDissableFunctions.IN := FALSE; END_IF  
			timDissableFunctions(IN:= , PT:= Lynus_Standards.Constants_General.tTimeDissableLynusFunctions, Q=> , ET=> );

(*-----------------------------------------------------------------------------Error ----------------------------------------------------------------------------*)

fbDIErrorPv(bInvers:= FALSE, bSignal=> );	

IF timDissableFunctions.Q THEN fbPv.bWarning := TRUE; fbPv.iWarningCode := 0; ELSE fbPv.bWarning := FALSE; END_IF 	
	IF fbDIErrorPv.bSignal OR Lynus_Standards.GVL_Energy.stNumberOfDevices.diNumberOfPvSystems > Constants_Energy.diMaxNumberOfPvSystems THEN fbPv.bError := TRUE; ELSE fbPv.bError := FALSE; END_IF 
		//Error Code
		IF Lynus_Standards.GVL_Energy.stNumberOfDevices.diNumberOfPvSystems > Constants_Energy.diMaxNumberOfPvSystems THEN fbPv.iErrorCode := 1; END_IF  
		IF fbDIErrorPv.bSignal THEN fbPv.iErrorCode := 0; END_IF 

fbPv(
	bEnable:= bEnable AND NOT timDissableFunctions.Q, 
	bError:= , 
	bWriteWithDelay:= TRUE, 
	iErrorCode:= , 
	iWarningCode:= , 
	lrTotalCounterEnergy_Consumption:= , 
	lrTotalCounterEnergy_Production:= , 
	lrCounterEnergyT1_Consumption:= , 
	lrCounterEnergyT2_Consumption:= , 
	lrCounterEnergyT1_Production:= , 
	lrCounterEnergyT2_Production:= , 
	lrPvPower:= Lynus_Standards.GVL_Energy.stDataElectricMeters[diNrOfEM_IN_PV].lrPower * 1000, 
	tTimDelayOutput:= T#5S, 
	stDataPvOut=> , 
	stDataPvOutDelay=> stDataPv);	
		
(*-----------------------------------------------------------Handle data to Global structure for the Pv system-----------------------------------------------------------------*)

CASE iStateGVLData OF
	
	0://Init Step
		byWaitInStep := 0;
			diCounterForGVL := 1;
	
	1://Wait for 4 Steps before clean al Data on GVL
		byWaitInStep := byWaitInStep + 1;
			IF byWaitInStep >= 4 AND fbNumberDevice.bNumberIsCalculatet THEN iStateGVLData := 2; END_IF
				//To much Devices, back to the Init step
				IF byWaitInStep >= 4 AND NOT fbNumberDevice.bNumberIsCalculatet THEN iStateGVLData := 0; END_IF	
			
	2://Clear all Data in GVL
		Lynus_Standards.GVL_Energy.stDataOfPvSystems[diCounterForGVL].bEnabled := FALSE;
			Lynus_Standards.GVL_Energy.stDataOfPvSystems[diCounterForGVL].byErrorWarning := 0;
				Lynus_Standards.GVL_Energy.stDataOfPvSystems[diCounterForGVL].lrPowerConsumption := 0;
					Lynus_Standards.GVL_Energy.stDataOfPvSystems[diCounterForGVL].lrPower := 0;
						Lynus_Standards.GVL_Energy.stDataOfPvSystems[diCounterForGVL].lrPowerProduction := 0;	
		
		diCounterForGVL := diCounterForGVL + 1;
			diCounterForGVL := LIMIT(0,diCounterForGVL,Constants_Energy.diMaxNumberOfPvSystems);
				//Back to the init step
				IF diCounterForGVL >= Constants_Energy.diMaxNumberOfPvSystems THEN iStateGVLData := 0; END_IF

END_CASE 	 

IF diNrOfPv_OUT > 0 AND fbNumberDevice.bNumberIsCalculatet THEN
	Lynus_Standards.GVL_Energy.stDataOfPvSystems[diNrOfPv_OUT].bEnabled := fbPv.stDataPvOut.bEnabled;
		Lynus_Standards.GVL_Energy.stDataOfPvSystems[diNrOfPv_OUT].byErrorWarning := fbPv.stDataPvOut.byErrorWarning;
			Lynus_Standards.GVL_Energy.stDataOfPvSystems[diNrOfPv_OUT].lrPowerConsumption := fbPv.stDataPvOut.lrPowerConsumption;
				Lynus_Standards.GVL_Energy.stDataOfPvSystems[diNrOfPv_OUT].lrPower := fbPv.stDataPvOut.lrPower;
					Lynus_Standards.GVL_Energy.stDataOfPvSystems[diNrOfPv_OUT].lrPowerProduction := fbPv.stDataPvOut.lrPowerProduction;
END_IF

(*----------------------------------------------------------Save persistent data----------------------------------------------------------------*)

arrPD[1](lrValue:= BOOL_TO_LREAL(bEnable), bEventBasedActive=> );
arrPD[2](lrValue:= BOOL_TO_LREAL(bPowerDataInvers), bEventBasedActive=> );
arrPD[3](lrValue:= DINT_TO_LREAL(diNrOfEM_IN_PV), bEventBasedActive=> );

END_FUNCTION_BLOCK

// ---- FBs/PV/FB_PV_Power_Ext_Input.TcPOU
FUNCTION_BLOCK FB_PV_Power_Ext_Input
VAR_INPUT PERSISTENT
	bEnable									: BOOL;													//Enable the Fuctionblock and his logic
END_VAR
VAR_INPUT
	bExtErrorPv								: BOOL;													//External Error for the Pv Function
	lrExtPvPower							: LREAL;												//External Pv power from a other Function or calculation in kW
	lrExtTotalCounterEnergy_Consumption		: LREAL;												//External Counter Value for Energy consumption with unit kWh
	lrExtTotalCounterEnergy_Production		: LREAL;												//External Counter Value for Energy production with unit kWh
	lrExtCounterEnergyT1_Consumption		: LREAL;												//External Counter Value for Energy consumption Tariff 1 with unit kWh
	lrExtCounterEnergyT2_Consumption		: LREAL;												//External Counter Value for Energy consumption Tariff 2 with unit kWh
	lrExtCounterEnergyT1_Production			: LREAL;												//External Counter Value for Energy production Tariff 1 with unit kWh
	lrExtCounterEnergyT2_Production			: LREAL;												//External Counter Value for Energy production Tariff 2 with unit kWh
END_VAR
VAR_OUTPUT
	stDataPv								: ST_PV_Output;											//{#lynus.ag#()} //Output Data Pv System
	diNrOfPv_OUT							: DINT;													//Active Number from the Pv system for using on other functions
END_VAR
VAR
	{attribute 'hide'}
	fbPv									: FB_PV_Production;										//Function block for Pv system
	{attribute 'hide'}
	fbNumberDevice							: FB_NumberOfDevice;									//Function block to calcualte the number of the Device
	fbDIErrorPv								: FB_XL1XXX_DI;											//Digital Input Error Pv System
	{attribute 'hide'}
	timDissableFunctions					: TON;													//Timer to dissable the Function after Lynus_Standards.Constants_General.tTimeDissableLynusFunctions Days without connection to the Lynus Cloud
	{attribute 'hide'}
	timResetConnectionOnGVL					: TON;													//Timer to try reset the connection Flag on the GVL. (When somebody delete the Connection Function and make only a onlinechange)
	{attribute 'hide'}
	fbPD									: FB_PersistentData_Number;								//Function to save persistent data 
	{attribute 'hide'}
	byWaitInStep							: BYTE;													//Wait in Step before start to clean data on PLC
	{attribute 'hide'}
	iStateGVLData							: INT;													//State machine to handle the data on the GVL
	{attribute 'hide'}
	diCounterForGVL							: DINT;													//Counter to clean old data on GVL
END_VAR

//Creator : Kai Ebensperger
//Company : Lynus AG
//Date : 08.06.2021
//Version : 1.0.0.0

//With this function block its possible to show the power data from a PV system.
//The Power and Error Data came from a other Function and can connect to the Inputs. The Function write the Data then on the Lynus GVL

//NOTE for diNr.....Designation => 
//_IN = Here Data come in from other Functions or go out to other functions about the GVL
//_OUT = Here Data go out to other functions about the GVL

(*-------------------------------------------------------------Calcualte the number of Pv System---------------------------------------------------------------*)

fbNumberDevice(
	diActualNumberOfDevices:= Lynus_Standards.GVL_Energy.stNumberOfDevices.diNumberOfPvSystems, 
	diMaxNumberOfDevices:= Constants_Energy.diMaxNumberOfPvSystems, 
	udiCounterOnlineChange:= TwinCAT_SystemInfoVarList._AppInfo.OnlineChangeCnt, 
	bNumberIsCalculatet=> , 
	bFPNumberIsCalculatet=> , 
	bOnlineChange=> , 
	diNumberForThisDevice=> diNrOfPv_OUT, 
	diNumberOfTotalDevices=> );

//Write new Numer on GVL
IF fbNumberDevice.bFPNumberIsCalculatet THEN
	Lynus_Standards.GVL_Energy.stNumberOfDevices.diNumberOfPvSystems := fbNumberDevice.diNumberOfTotalDevices;	
END_IF 

//Delete old Number on GVL
IF fbNumberDevice.bOnlineChange THEN 
	Lynus_Standards.GVL_Energy.stNumberOfDevices.diNumberOfPvSystems := diNrOfPv_OUT;	
		iStateGVLData := 1; 
END_IF	

(*-------------------------------------------------------------Service from Backend is ready and check the connection to backen for dissabel/enable Function---------------------------------------------------------------*)

//Try to reset the variable for connection on the GVL. When all is normal then the Lynus Mqtt connection function set this variable to true in the next cycle
//When we have no connection to the backend then after Lynus_Standards.Constants_General.tTimeDissableLynusFunctions days the Function is dissabled with all of his functionalities
timResetConnectionOnGVL(IN:= NOT timResetConnectionOnGVL.Q, PT:= T#1H, Q=> , ET=> );
	IF timResetConnectionOnGVL.Q THEN Lynus_Standards.GVL_Communicator.bStateConnectionToEnableFunctions := FALSE; END_IF
		IF NOT Lynus_Standards.GVL_Communicator.bStateConnectionToEnableFunctions THEN timDissableFunctions.IN := TRUE; ELSE timDissableFunctions.IN := FALSE; END_IF  
			timDissableFunctions(IN:= , PT:= Lynus_Standards.Constants_General.tTimeDissableLynusFunctions, Q=> , ET=> );

(*-----------------------------------------------------------------------------Error ----------------------------------------------------------------------------*)

fbDIErrorPv(bInvers:= FALSE, bSignal=> );	

IF timDissableFunctions.Q THEN fbPv.bWarning := TRUE; fbPv.iWarningCode := 0; ELSE fbPv.bWarning := FALSE; END_IF 	
	IF fbDIErrorPv.bSignal OR Lynus_Standards.GVL_Energy.stNumberOfDevices.diNumberOfPvSystems > Constants_Energy.diMaxNumberOfPvSystems OR bExtErrorPv THEN fbPv.bError := TRUE; ELSE fbPv.bError := FALSE; END_IF 
		//Error Code
		IF Lynus_Standards.GVL_Energy.stNumberOfDevices.diNumberOfPvSystems > Constants_Energy.diMaxNumberOfPvSystems THEN fbPv.iErrorCode := 1; END_IF  
		IF fbDIErrorPv.bSignal OR bExtErrorPv THEN fbPv.iErrorCode := 0; END_IF 

fbPv(
	bEnable:= bEnable AND NOT timDissableFunctions.Q, 
	bError:= , 
	bWriteWithDelay:= TRUE, 
	iErrorCode:= , 
	iWarningCode:= , 
	lrTotalCounterEnergy_Consumption:= lrExtTotalCounterEnergy_Consumption * 1000, 
	lrTotalCounterEnergy_Production:= lrExtTotalCounterEnergy_Production * 1000, 
	lrCounterEnergyT1_Consumption:= lrExtCounterEnergyT1_Consumption * 1000, 
	lrCounterEnergyT2_Consumption:= lrExtCounterEnergyT2_Consumption * 1000, 
	lrCounterEnergyT1_Production:= lrExtCounterEnergyT1_Production * 1000, 
	lrCounterEnergyT2_Production:= lrExtCounterEnergyT2_Production * 1000, 
	lrPvPower:= lrExtPvPower * 1000, 
	tTimDelayOutput:= T#5S, 
	stDataPvOut=> , 
	stDataPvOutDelay=> stDataPv);	
		
(*-----------------------------------------------------------Handle data to Global structure for the Pv system-----------------------------------------------------------------*)

CASE iStateGVLData OF
	
	0://Init Step
		byWaitInStep := 0;
			diCounterForGVL := 1;
	
	1://Wait for 4 Steps before clean al Data on GVL
		byWaitInStep := byWaitInStep + 1;
			IF byWaitInStep >= 4 AND fbNumberDevice.bNumberIsCalculatet THEN iStateGVLData := 2; END_IF
				//To much Devices, back to the Init step
				IF byWaitInStep >= 4 AND NOT fbNumberDevice.bNumberIsCalculatet THEN iStateGVLData := 0; END_IF	
			
	2://Clear all Data in GVL
		Lynus_Standards.GVL_Energy.stDataOfPvSystems[diCounterForGVL].bEnabled := FALSE;
			Lynus_Standards.GVL_Energy.stDataOfPvSystems[diCounterForGVL].byErrorWarning := 0;
				Lynus_Standards.GVL_Energy.stDataOfPvSystems[diCounterForGVL].lrPowerConsumption := 0;
					Lynus_Standards.GVL_Energy.stDataOfPvSystems[diCounterForGVL].lrPower := 0;
						Lynus_Standards.GVL_Energy.stDataOfPvSystems[diCounterForGVL].lrPowerProduction := 0;	
		
		diCounterForGVL := diCounterForGVL + 1;
			diCounterForGVL := LIMIT(0,diCounterForGVL,Constants_Energy.diMaxNumberOfPvSystems);
				//Back to the init step
				IF diCounterForGVL >= Constants_Energy.diMaxNumberOfPvSystems THEN iStateGVLData := 0; END_IF

END_CASE 	 

IF diNrOfPv_OUT > 0 AND fbNumberDevice.bNumberIsCalculatet THEN
	Lynus_Standards.GVL_Energy.stDataOfPvSystems[diNrOfPv_OUT].bEnabled := fbPv.stDataPvOut.bEnabled;
		Lynus_Standards.GVL_Energy.stDataOfPvSystems[diNrOfPv_OUT].byErrorWarning := fbPv.stDataPvOut.byErrorWarning;
			Lynus_Standards.GVL_Energy.stDataOfPvSystems[diNrOfPv_OUT].lrPowerConsumption := fbPv.stDataPvOut.lrPowerConsumption;
				Lynus_Standards.GVL_Energy.stDataOfPvSystems[diNrOfPv_OUT].lrPower := fbPv.stDataPvOut.lrPower;
					Lynus_Standards.GVL_Energy.stDataOfPvSystems[diNrOfPv_OUT].lrPowerProduction := fbPv.stDataPvOut.lrPowerProduction;
END_IF

(*----------------------------------------------------------Save persistent data----------------------------------------------------------------*)

fbPD(lrValue:= BOOL_TO_LREAL(bEnable), bEventBasedActive=> );

END_FUNCTION_BLOCK

// ---- FBs/Setpoint Optimizer/FB_SPOpt_AirSystem.TcPOU
{attribute 'hide_all_locals'}
FUNCTION_BLOCK FB_SPOpt_AirSystem
VAR_INPUT PERSISTENT
	bEnable							: BOOL;									//Enable or dissable thsi Function
END_VAR
VAR_INPUT
	byStateSystemIn					: BYTE;									//Actual State from the System. 0 = off, 1 = on
	rFlowAirTempIn					: REAL;									//Actual Flow Air Temperature
	rReturnAirTempIn				: REAL;									//Actual Return Air Temperature
	rInToOutAirTempIn				: REAL;									//Actual outdoor air flow temperature
	rOutToInAirTempIn				: REAL;									//Actual indoor air flow temperature
END_VAR
VAR_OUTPUT
	bError							: BOOL;									//Error from this Fuction
	byStateSystemOut				: BYTE;									//{#lynus.ag#()} //State from the System. 0 = off, 1 = on	
	rFlowAirTempOut					: REAL;									//{#lynus.ag#()} //Flow Air Temperature to send to the Backend Service.
	rReturnAirTempOut				: REAL;									//{#lynus.ag#()} //Return Air Temperature to send to the Backend Service.
	rInToOutAirTempOut				: REAL;									//{#lynus.ag#()} //Outdoor air flow temperature to send to the Backend Service.
	rOutToInAirTempOut				: REAL;									//{#lynus.ag#()} //Indoor air flow temperature to send to the Backend Service.
	diNrOfSPOpt_OUT					: DINT;									//Active Number from Setpoint Optimizer for using on other functions
END_VAR
VAR
	fbNumberDevice					: FB_NumberOfDevice;					//Function block to calcualte the number of the Device
	timDissableFunctions			: TON;									//Timer to dissable the Function after Lynus_Standards.Constants_General.tTimeDissableLynusFunctions Days without connection to the Lynus Cloud
	timResetConnectionOnGVL			: TON;									//Timer to try reset the connection Flag on the GVL. (When somebody delete the Connection Function and make only a onlinechange)
END_VAR

//Creator : Kai Ebensperger
//Company : Lynus AG
//Date : 03.12.2021
//Version : 1.0.0.0

//This Function is a Help Function for the Setpoint Optimizer on our Backend System
//Here we can read in the neccessary Values for a Air System from a external Service and can send then to the Backend System for optimizing
//Its Helpfull if we work with the TMC File

(*----------------------------------------------------------------------------------------Limits---------------------------------------------------------------------------------------------------------------*)

byStateSystemIn := LIMIT(0,byStateSystemIn,1);
	rFlowAirTempIn := LIMIT(-30,rFlowAirTempIn,150);
		rReturnAirTempIn := LIMIT(-30,rReturnAirTempIn,150);
			rInToOutAirTempIn := LIMIT(-30,rInToOutAirTempIn,150);
				rOutToInAirTempIn := LIMIT(-30,rOutToInAirTempIn,150);

(*-------------------------------------------------------------Calcualte the number of SP Opttimizer---------------------------------------------------------------*)

fbNumberDevice(
	diActualNumberOfDevices:= Lynus_Standards.GVL_Energy.stNumberOfDevices.diNumberOfSetPointOpt, 
	diMaxNumberOfDevices:= Constants_Energy.diMaxNumberOfSetPointOpt, 
	udiCounterOnlineChange:= TwinCAT_SystemInfoVarList._AppInfo.OnlineChangeCnt, 
	bNumberIsCalculatet=> , 
	bFPNumberIsCalculatet=> , 
	bOnlineChange=> , 
	diNumberForThisDevice=> diNrOfSPOpt_OUT, 
	diNumberOfTotalDevices=> );

//Write new Numer on GVL
IF fbNumberDevice.bFPNumberIsCalculatet THEN
	Lynus_Standards.GVL_Energy.stNumberOfDevices.diNumberOfSetPointOpt := fbNumberDevice.diNumberOfTotalDevices;	
END_IF 

//Delete old Number on GVL
IF fbNumberDevice.bOnlineChange THEN 
	Lynus_Standards.GVL_Energy.stNumberOfDevices.diNumberOfSetPointOpt := diNrOfSPOpt_OUT;
END_IF				
				
(*-------------------------------------------------------------Service from Backend is ready and check the connection to backen for dissabel/enable EMS Function---------------------------------------------------------------*)

//Try to reset the variable for connection on the GVL. When all is normal then the Lynus Mqtt connection function set this variable to true in the next cycle
//When we have no connection to the backend or no HB from the Service then after Lynus_Standards.Constants_General.tTimeDissableLynusFunctions days the EMS is dissabled with all of his functionalities
timResetConnectionOnGVL(IN:= NOT timResetConnectionOnGVL.Q, PT:= T#1H, Q=> , ET=> );
	IF timResetConnectionOnGVL.Q THEN Lynus_Standards.GVL_Communicator.bStateConnectionToEnableFunctions := FALSE; END_IF
		IF NOT Lynus_Standards.GVL_Communicator.bStateConnectionToEnableFunctions THEN timDissableFunctions.IN := TRUE; ELSE timDissableFunctions.IN := FALSE; END_IF  
			timDissableFunctions(IN:= , PT:= Lynus_Standards.Constants_General.tTimeDissableLynusFunctions, Q=> , ET=> );

(*------------------------------------------------------------------Error----------------------------------------------------------------------------*)	

IF Lynus_Standards.GVL_Energy.stNumberOfDevices.diNumberOfSetPointOpt > Constants_Energy.diMaxNumberOfSetPointOpt THEN bError := TRUE; ELSE bError := FALSE; END_IF 			
			
(*-------------------------------------------------------------------------------------In to Out---------------------------------------------------------------------------------------*)

byStateSystemOut := byStateSystemIn;
	rFlowAirTempOut := rFlowAirTempIn;
		rReturnAirTempOut := rReturnAirTempIn;	
			rInToOutAirTempOut := rInToOutAirTempIn;
				rOutToInAirTempOut := rOutToInAirTempIn;		

IF NOT bEnable OR timDissableFunctions.Q OR Lynus_Standards.GVL_Energy.stNumberOfDevices.diNumberOfSetPointOpt > Constants_Energy.diMaxNumberOfSetPointOpt THEN
	byStateSystemOut := 0;	
END_IF

END_FUNCTION_BLOCK

